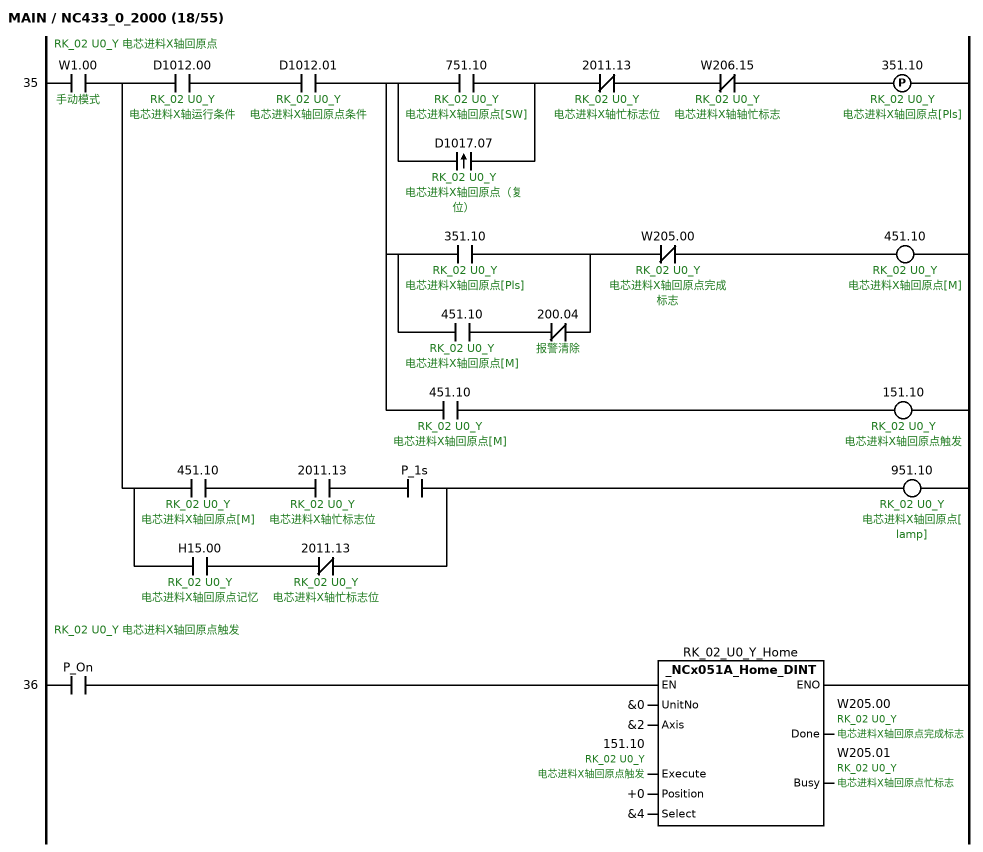
; [picture p72: MAIN / NC433_0_2000, rungs 35-36]
; rung 35: RK_02 U0_Y 电芯进料X轴回原点
LD W1.00  ; 手动模式
OUT TR0
AND D1012.00  ; RK_02 U0_Y 电芯进料X轴运行条件
AND D1012.01  ; RK_02 U0_Y 电芯进料X轴回原点条件
OUT TR1
LD 751.10  ; RK_02 U0_Y 电芯进料X轴回原点[SW]
@OR D1017.07  ; RK_02 U0_Y 电芯进料X轴回原点（复位）
ANDLD
ANDNOT 2011.13  ; RK_02 U0_Y 电芯进料X轴忙标志位
ANDNOT W206.15  ; RK_02 U0_Y 电芯进料X轴轴忙标志
DIFU(013) 351.10  ; RK_02 U0_Y 电芯进料X轴回原点[Pls]
LD TR1
LD 351.10  ; RK_02 U0_Y 电芯进料X轴回原点[Pls]
LD 451.10  ; RK_02 U0_Y 电芯进料X轴回原点[M]
ANDNOT 200.04  ; 报警清除
ORLD
ANDLD
ANDNOT W205.00  ; RK_02 U0_Y 电芯进料X轴回原点完成标志
OUT 451.10  ; RK_02 U0_Y 电芯进料X轴回原点[M]
LD TR1
AND 451.10  ; RK_02 U0_Y 电芯进料X轴回原点[M]
OUT 151.10  ; RK_02 U0_Y 电芯进料X轴回原点触发
LD TR0
LD 451.10  ; RK_02 U0_Y 电芯进料X轴回原点[M]
AND 2011.13  ; RK_02 U0_Y 电芯进料X轴忙标志位
AND P_1s
LD H15.00  ; RK_02 U0_Y 电芯进料X轴回原点记忆
ANDNOT 2011.13  ; RK_02 U0_Y 电芯进料X轴忙标志位
ORLD
ANDLD
OUT 951.10  ; RK_02 U0_Y 电芯进料X轴回原点[lamp]
; rung 36: RK_02 U0_Y 电芯进料X轴回原点触发
LD P_On
CALL RK_02_U0_Y_Home : _NCx051A_Home_DINT (UnitNo := &0, Axis := &2, Execute := 151.10, Position := +0, Select := &4, Done => W205.00, Busy => W205.01)  ; RK_02 U0_Y 电芯进料X轴回原点触发, RK_02 U0_Y 电芯进料X轴回原点完成标志, RK_02 U0_Y 电芯进料X轴回原点忙标志

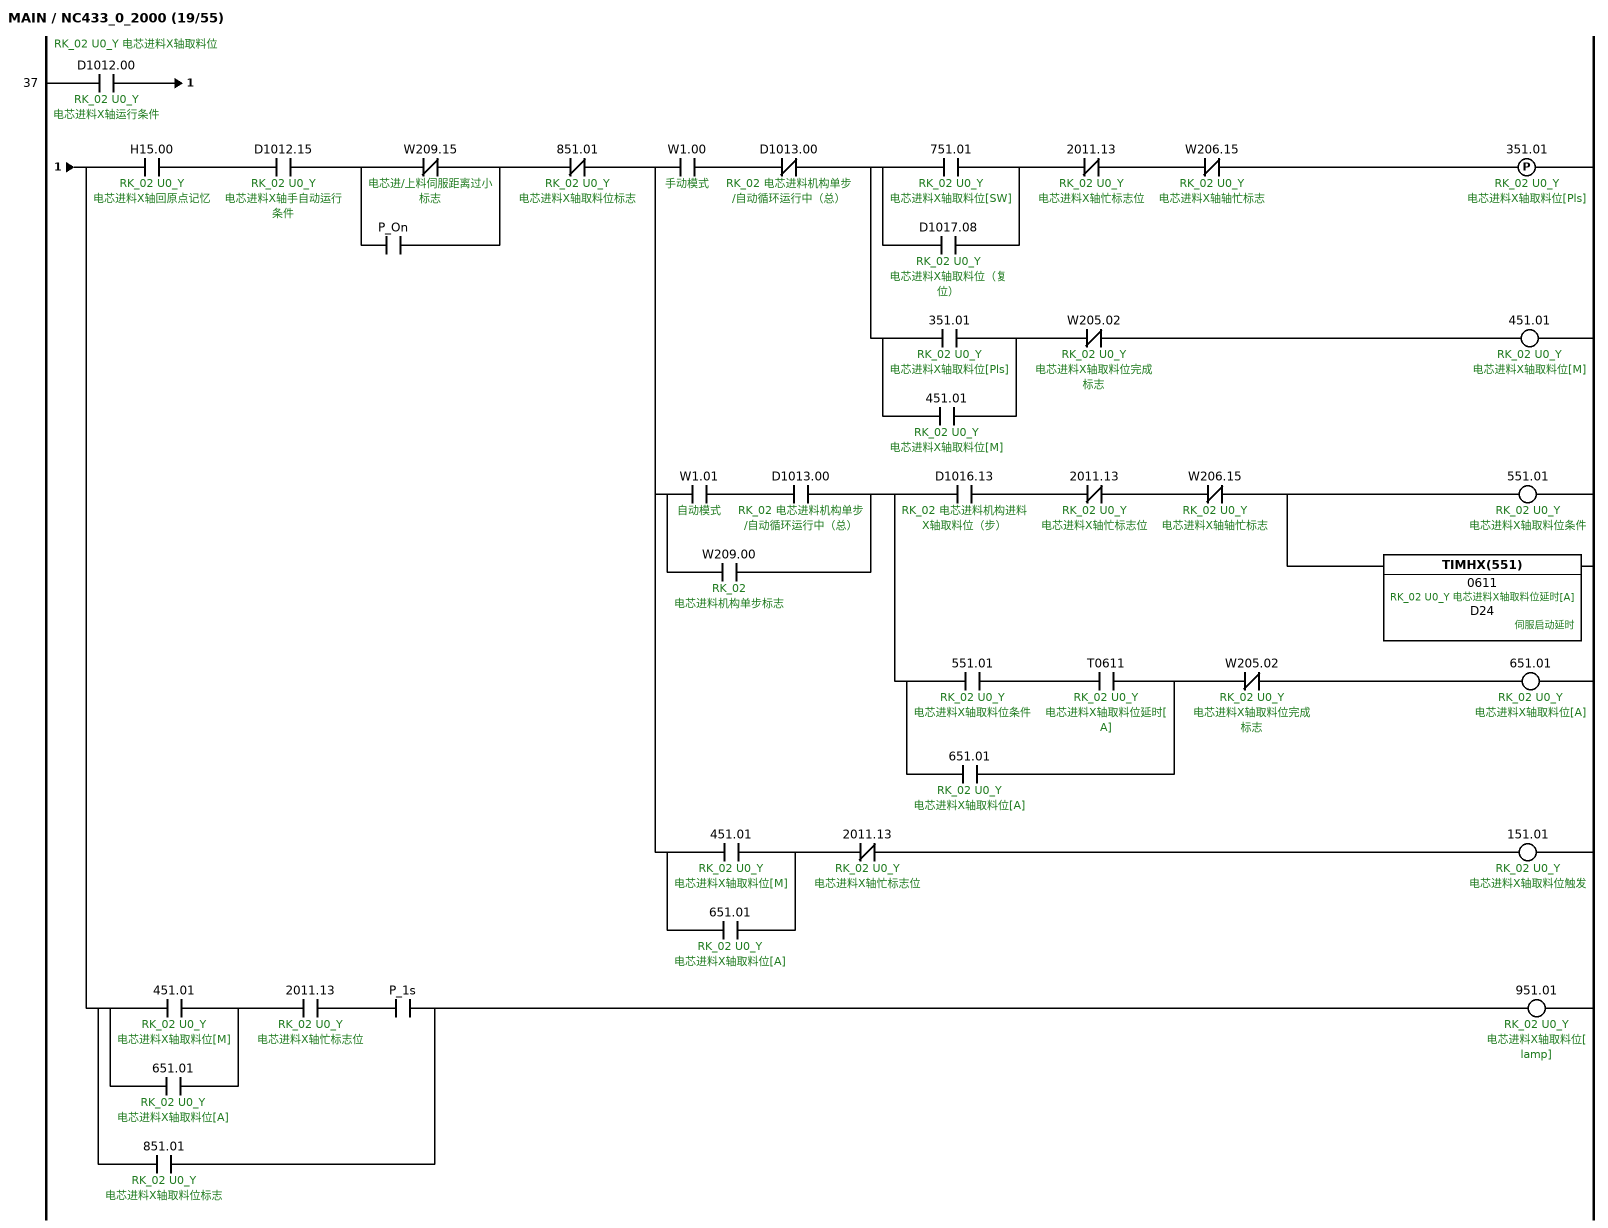
; rung 37: RK_02 U0_Y 电芯进料X轴取料位
LD D1012.00  ; RK_02 U0_Y 电芯进料X轴运行条件
OUT TR0
AND H15.00  ; RK_02 U0_Y 电芯进料X轴回原点记忆
AND D1012.15  ; RK_02 U0_Y 电芯进料X轴手自动运行条件
LDNOT W209.15  ; 电芯进/上料伺服距离过小标志
OR P_On
ANDLD
ANDNOT 851.01  ; RK_02 U0_Y 电芯进料X轴取料位标志
OUT TR1
AND W1.00  ; 手动模式
ANDNOT D1013.00  ; RK_02 电芯进料机构单步/自动循环运行中（总）
OUT TR2
LD 751.01  ; RK_02 U0_Y 电芯进料X轴取料位[SW]
OR D1017.08  ; RK_02 U0_Y 电芯进料X轴取料位（复位）
ANDLD
ANDNOT 2011.13  ; RK_02 U0_Y 电芯进料X轴忙标志位
ANDNOT W206.15  ; RK_02 U0_Y 电芯进料X轴轴忙标志
DIFU(013) 351.01  ; RK_02 U0_Y 电芯进料X轴取料位[Pls]
LD TR2
LD 351.01  ; RK_02 U0_Y 电芯进料X轴取料位[Pls]
OR 451.01  ; RK_02 U0_Y 电芯进料X轴取料位[M]
ANDLD
ANDNOT W205.02  ; RK_02 U0_Y 电芯进料X轴取料位完成标志
OUT 451.01  ; RK_02 U0_Y 电芯进料X轴取料位[M]
LD TR1
LD W1.01  ; 自动模式
AND D1013.00  ; RK_02 电芯进料机构单步/自动循环运行中（总）
OR W209.00  ; RK_02  电芯进料机构单步标志
ANDLD
OUT TR2
AND D1016.13  ; RK_02 电芯进料机构进料X轴取料位（步）
ANDNOT 2011.13  ; RK_02 U0_Y 电芯进料X轴忙标志位
ANDNOT W206.15  ; RK_02 U0_Y 电芯进料X轴轴忙标志
OUT 551.01  ; RK_02 U0_Y 电芯进料X轴取料位条件
TIMHX(551) 0611 D24  ; 伺服启动延时, RK_02 U0_Y 电芯进料X轴取料位延时[A]
LD TR2
LD 551.01  ; RK_02 U0_Y 电芯进料X轴取料位条件
AND T0611  ; RK_02 U0_Y 电芯进料X轴取料位延时[A]
OR 651.01  ; RK_02 U0_Y 电芯进料X轴取料位[A]
ANDLD
ANDNOT W205.02  ; RK_02 U0_Y 电芯进料X轴取料位完成标志
OUT 651.01  ; RK_02 U0_Y 电芯进料X轴取料位[A]
LD TR1
LD 451.01  ; RK_02 U0_Y 电芯进料X轴取料位[M]
OR 651.01  ; RK_02 U0_Y 电芯进料X轴取料位[A]
ANDLD
ANDNOT 2011.13  ; RK_02 U0_Y 电芯进料X轴忙标志位
OUT 151.01  ; RK_02 U0_Y 电芯进料X轴取料位触发
LD TR0
LD 451.01  ; RK_02 U0_Y 电芯进料X轴取料位[M]
OR 651.01  ; RK_02 U0_Y 电芯进料X轴取料位[A]
AND 2011.13  ; RK_02 U0_Y 电芯进料X轴忙标志位
AND P_1s
OR 851.01  ; RK_02 U0_Y 电芯进料X轴取料位标志
ANDLD
OUT 951.01  ; RK_02 U0_Y 电芯进料X轴取料位[lamp]

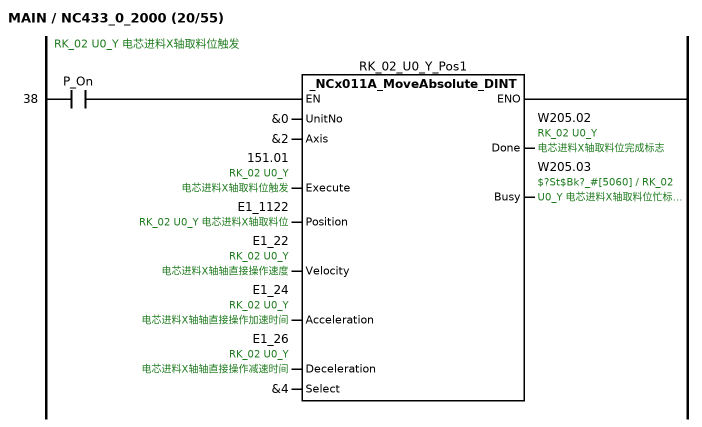
; rung 38: RK_02 U0_Y 电芯进料X轴取料位触发
LD P_On
CALL RK_02_U0_Y_Pos1 : _NCx011A_MoveAbsolute_DINT (UnitNo := &0, Axis := &2, Execute := 151.01, Position := E1_1122, Velocity := E1_22, Acceleration := E1_24, Deceleration := E1_26, Select := &4, Done => W205.02, Busy => W205.03)  ; RK_02 U0_Y 电芯进料X轴取料位触发, RK_02 U0_Y 电芯进料X轴取料位, RK_02 U0_Y 电芯进料X轴轴直接操作速度, RK_02 U0_Y 电芯进料X轴轴直接操作加速时间, RK_02 U0_Y 电芯进料X轴轴直接操作减速时间, RK_02 U0_Y 电芯进料X轴取料位完成标志, $?St$Bk?_#[5060] / RK_02 U0_Y 电芯进料X轴取料位忙标志 / $?St$Bk?_#[5060]

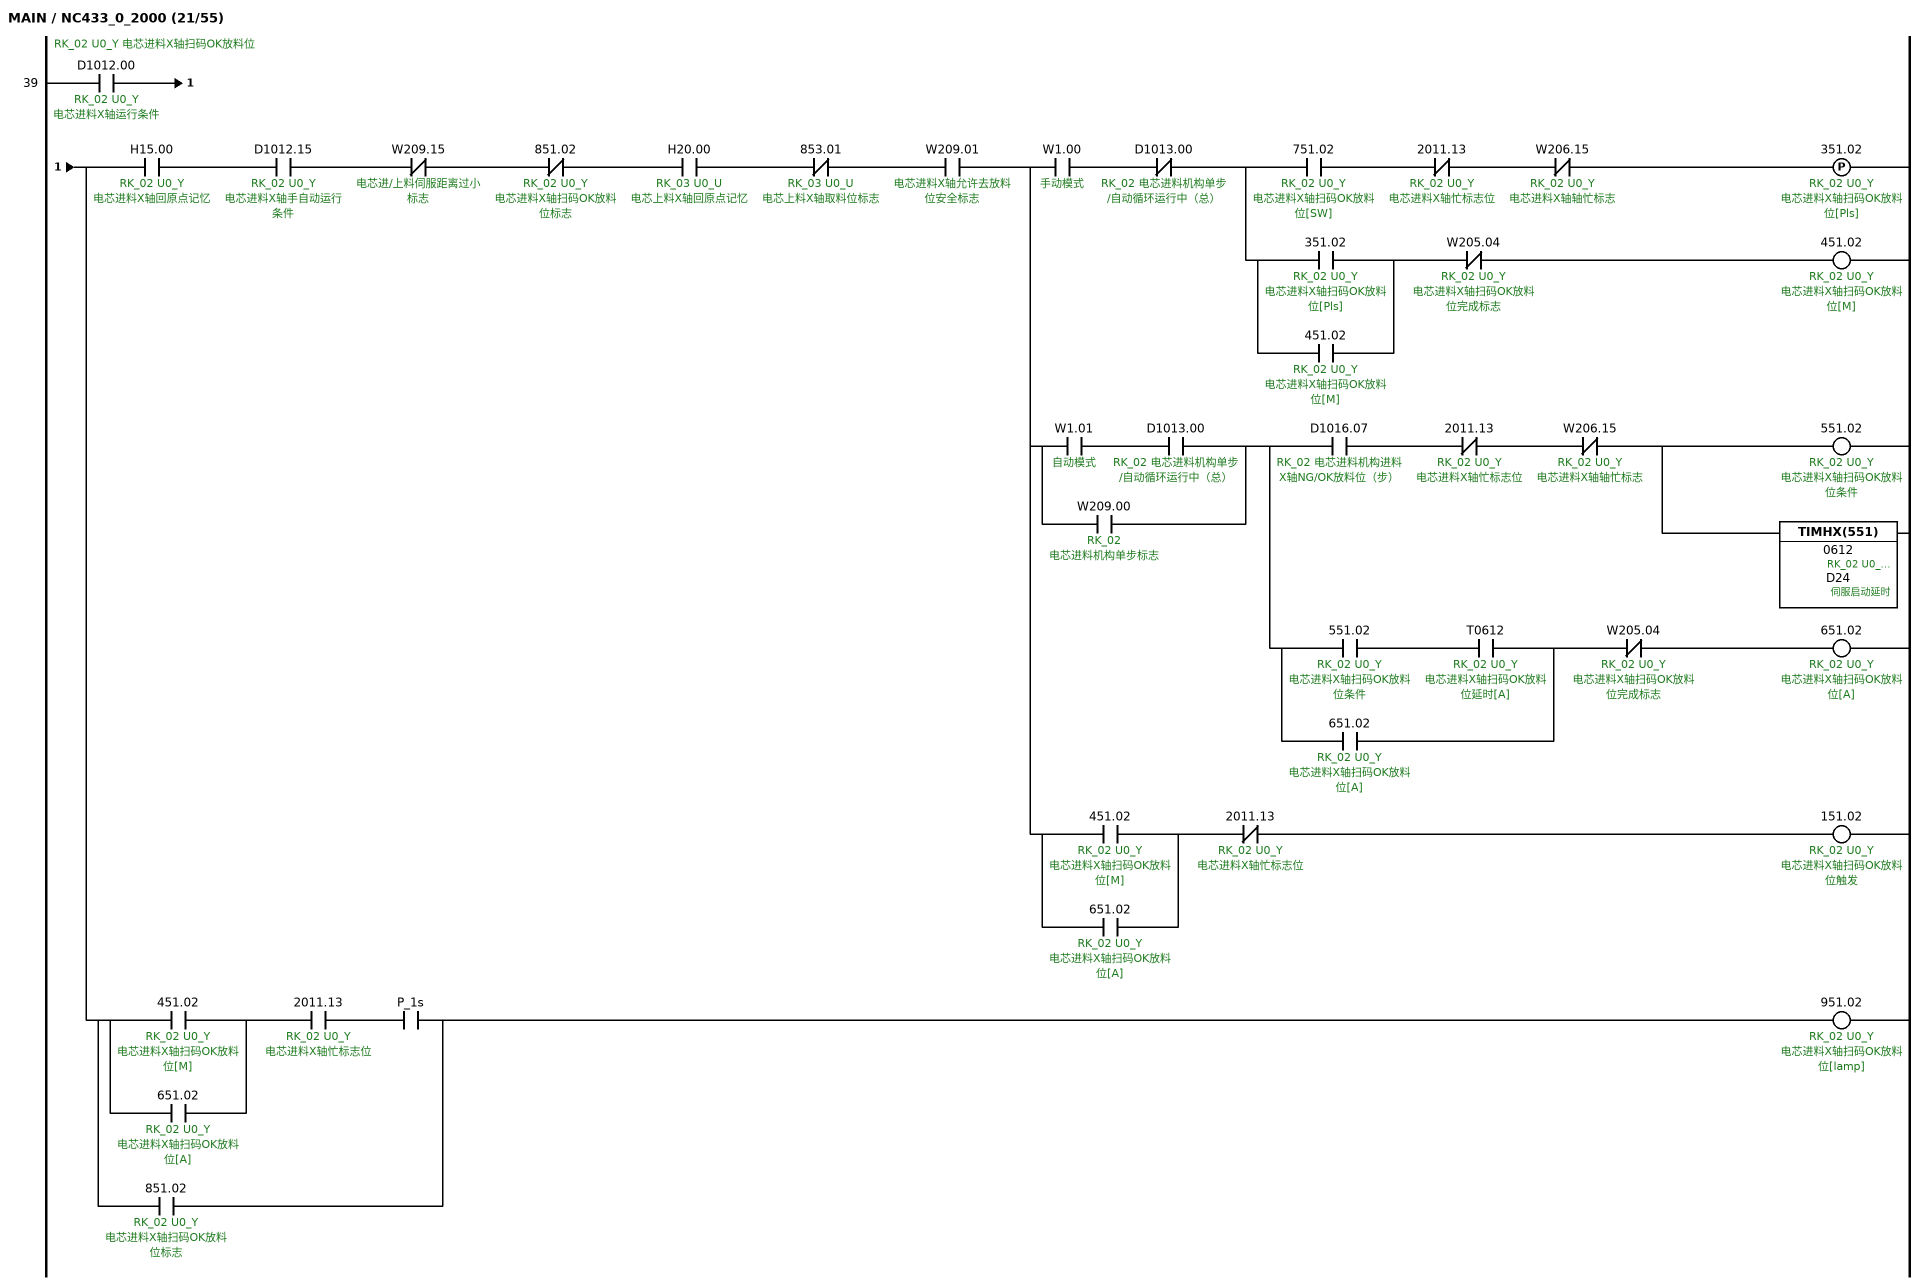
; rung 39: RK_02 U0_Y 电芯进料X轴扫码OK放料位
LD D1012.00  ; RK_02 U0_Y 电芯进料X轴运行条件
OUT TR0
AND H15.00  ; RK_02 U0_Y 电芯进料X轴回原点记忆
AND D1012.15  ; RK_02 U0_Y 电芯进料X轴手自动运行条件
ANDNOT W209.15  ; 电芯进/上料伺服距离过小标志
ANDNOT 851.02  ; RK_02 U0_Y 电芯进料X轴扫码OK放料位标志
AND H20.00  ; RK_03 U0_U 电芯上料X轴回原点记忆
ANDNOT 853.01  ; RK_03 U0_U 电芯上料X轴取料位标志
AND W209.01  ; 电芯进料X轴允许去放料位安全标志
OUT TR1
AND W1.00  ; 手动模式
ANDNOT D1013.00  ; RK_02 电芯进料机构单步/自动循环运行中（总）
OUT TR2
AND 751.02  ; RK_02 U0_Y 电芯进料X轴扫码OK放料位[SW]
ANDNOT 2011.13  ; RK_02 U0_Y 电芯进料X轴忙标志位
ANDNOT W206.15  ; RK_02 U0_Y 电芯进料X轴轴忙标志
DIFU(013) 351.02  ; RK_02 U0_Y 电芯进料X轴扫码OK放料位[Pls]
LD TR2
LD 351.02  ; RK_02 U0_Y 电芯进料X轴扫码OK放料位[Pls]
OR 451.02  ; RK_02 U0_Y 电芯进料X轴扫码OK放料位[M]
ANDLD
ANDNOT W205.04  ; RK_02 U0_Y 电芯进料X轴扫码OK放料位完成标志
OUT 451.02  ; RK_02 U0_Y 电芯进料X轴扫码OK放料位[M]
LD TR1
LD W1.01  ; 自动模式
AND D1013.00  ; RK_02 电芯进料机构单步/自动循环运行中（总）
OR W209.00  ; RK_02  电芯进料机构单步标志
ANDLD
OUT TR2
AND D1016.07  ; RK_02 电芯进料机构进料X轴NG/OK放料位（步）
ANDNOT 2011.13  ; RK_02 U0_Y 电芯进料X轴忙标志位
ANDNOT W206.15  ; RK_02 U0_Y 电芯进料X轴轴忙标志
OUT 551.02  ; RK_02 U0_Y 电芯进料X轴扫码OK放料位条件
TIMHX(551) 0612 D24  ; 伺服启动延时, RK_02 U0_Y 电芯进料X轴扫码OK放料位延时[A]
LD TR2
LD 551.02  ; RK_02 U0_Y 电芯进料X轴扫码OK放料位条件
AND T0612  ; RK_02 U0_Y 电芯进料X轴扫码OK放料位延时[A]
OR 651.02  ; RK_02 U0_Y 电芯进料X轴扫码OK放料位[A]
ANDLD
ANDNOT W205.04  ; RK_02 U0_Y 电芯进料X轴扫码OK放料位完成标志
OUT 651.02  ; RK_02 U0_Y 电芯进料X轴扫码OK放料位[A]
LD TR1
LD 451.02  ; RK_02 U0_Y 电芯进料X轴扫码OK放料位[M]
OR 651.02  ; RK_02 U0_Y 电芯进料X轴扫码OK放料位[A]
ANDLD
ANDNOT 2011.13  ; RK_02 U0_Y 电芯进料X轴忙标志位
OUT 151.02  ; RK_02 U0_Y 电芯进料X轴扫码OK放料位触发
LD TR0
LD 451.02  ; RK_02 U0_Y 电芯进料X轴扫码OK放料位[M]
OR 651.02  ; RK_02 U0_Y 电芯进料X轴扫码OK放料位[A]
AND 2011.13  ; RK_02 U0_Y 电芯进料X轴忙标志位
AND P_1s
OR 851.02  ; RK_02 U0_Y 电芯进料X轴扫码OK放料位标志
ANDLD
OUT 951.02  ; RK_02 U0_Y 电芯进料X轴扫码OK放料位[lamp]

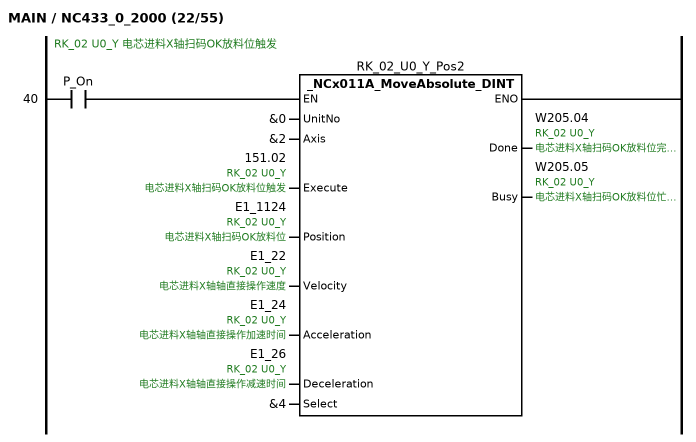
; rung 40: RK_02 U0_Y 电芯进料X轴扫码OK放料位触发
LD P_On
CALL RK_02_U0_Y_Pos2 : _NCx011A_MoveAbsolute_DINT (UnitNo := &0, Axis := &2, Execute := 151.02, Position := E1_1124, Velocity := E1_22, Acceleration := E1_24, Deceleration := E1_26, Select := &4, Done => W205.04, Busy => W205.05)  ; RK_02 U0_Y 电芯进料X轴扫码OK放料位触发, RK_02 U0_Y 电芯进料X轴扫码OK放料位, RK_02 U0_Y 电芯进料X轴轴直接操作速度, RK_02 U0_Y 电芯进料X轴轴直接操作加速时间, RK_02 U0_Y 电芯进料X轴轴直接操作减速时间, RK_02 U0_Y 电芯进料X轴扫码OK放料位完成标志, RK_02 U0_Y 电芯进料X轴扫码OK放料位忙标志

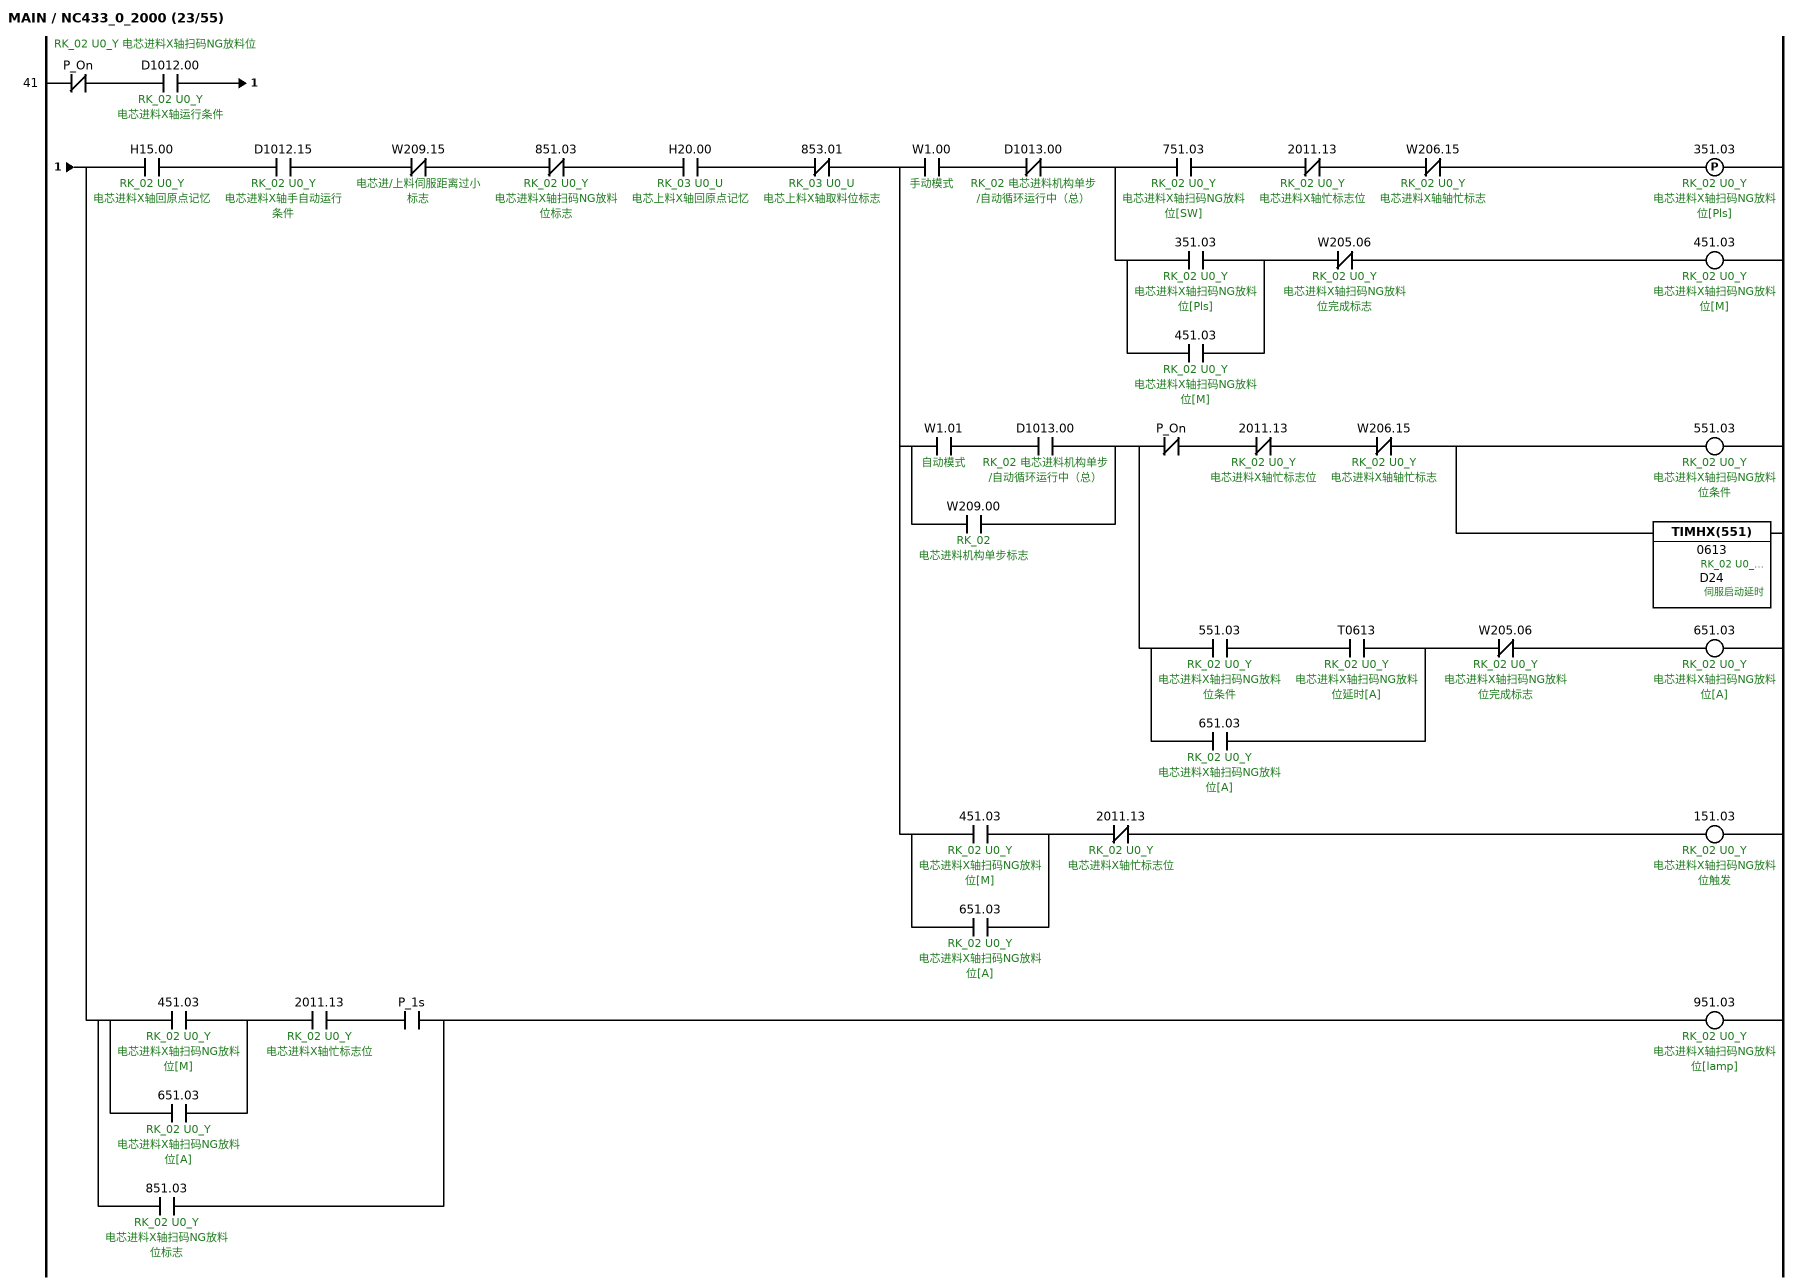
; rung 41: RK_02 U0_Y 电芯进料X轴扫码NG放料位
LDNOT P_On
AND D1012.00  ; RK_02 U0_Y 电芯进料X轴运行条件
OUT TR0
AND H15.00  ; RK_02 U0_Y 电芯进料X轴回原点记忆
AND D1012.15  ; RK_02 U0_Y 电芯进料X轴手自动运行条件
ANDNOT W209.15  ; 电芯进/上料伺服距离过小标志
ANDNOT 851.03  ; RK_02 U0_Y 电芯进料X轴扫码NG放料位标志
AND H20.00  ; RK_03 U0_U 电芯上料X轴回原点记忆
ANDNOT 853.01  ; RK_03 U0_U 电芯上料X轴取料位标志  // 或者改为“RK_03 U0_U 电芯上料X轴当前值”>“最小安全设定值”
OUT TR1
AND W1.00  ; 手动模式
ANDNOT D1013.00  ; RK_02 电芯进料机构单步/自动循环运行中（总）
OUT TR2
AND 751.03  ; RK_02 U0_Y 电芯进料X轴扫码NG放料位[SW]
ANDNOT 2011.13  ; RK_02 U0_Y 电芯进料X轴忙标志位
ANDNOT W206.15  ; RK_02 U0_Y 电芯进料X轴轴忙标志
DIFU(013) 351.03  ; RK_02 U0_Y 电芯进料X轴扫码NG放料位[Pls]
LD TR2
LD 351.03  ; RK_02 U0_Y 电芯进料X轴扫码NG放料位[Pls]
OR 451.03  ; RK_02 U0_Y 电芯进料X轴扫码NG放料位[M]
ANDLD
ANDNOT W205.06  ; RK_02 U0_Y 电芯进料X轴扫码NG放料位完成标志
OUT 451.03  ; RK_02 U0_Y 电芯进料X轴扫码NG放料位[M]
LD TR1
LD W1.01  ; 自动模式
AND D1013.00  ; RK_02 电芯进料机构单步/自动循环运行中（总）
OR W209.00  ; RK_02  电芯进料机构单步标志
ANDLD
OUT TR2
ANDNOT P_On  // RK_02 U0_Y 电芯进料X轴扫码NG放料位（步）
ANDNOT 2011.13  ; RK_02 U0_Y 电芯进料X轴忙标志位
ANDNOT W206.15  ; RK_02 U0_Y 电芯进料X轴轴忙标志
OUT 551.03  ; RK_02 U0_Y 电芯进料X轴扫码NG放料位条件
TIMHX(551) 0613 D24  ; 伺服启动延时, RK_02 U0_Y 电芯进料X轴扫码NG放料位延时[A]
LD TR2
LD 551.03  ; RK_02 U0_Y 电芯进料X轴扫码NG放料位条件
AND T0613  ; RK_02 U0_Y 电芯进料X轴扫码NG放料位延时[A]
OR 651.03  ; RK_02 U0_Y 电芯进料X轴扫码NG放料位[A]
ANDLD
ANDNOT W205.06  ; RK_02 U0_Y 电芯进料X轴扫码NG放料位完成标志
OUT 651.03  ; RK_02 U0_Y 电芯进料X轴扫码NG放料位[A]
LD TR1
LD 451.03  ; RK_02 U0_Y 电芯进料X轴扫码NG放料位[M]
OR 651.03  ; RK_02 U0_Y 电芯进料X轴扫码NG放料位[A]
ANDLD
ANDNOT 2011.13  ; RK_02 U0_Y 电芯进料X轴忙标志位
OUT 151.03  ; RK_02 U0_Y 电芯进料X轴扫码NG放料位触发
LD TR0
LD 451.03  ; RK_02 U0_Y 电芯进料X轴扫码NG放料位[M]
OR 651.03  ; RK_02 U0_Y 电芯进料X轴扫码NG放料位[A]
AND 2011.13  ; RK_02 U0_Y 电芯进料X轴忙标志位
AND P_1s
OR 851.03  ; RK_02 U0_Y 电芯进料X轴扫码NG放料位标志
ANDLD
OUT 951.03  ; RK_02 U0_Y 电芯进料X轴扫码NG放料位[lamp]

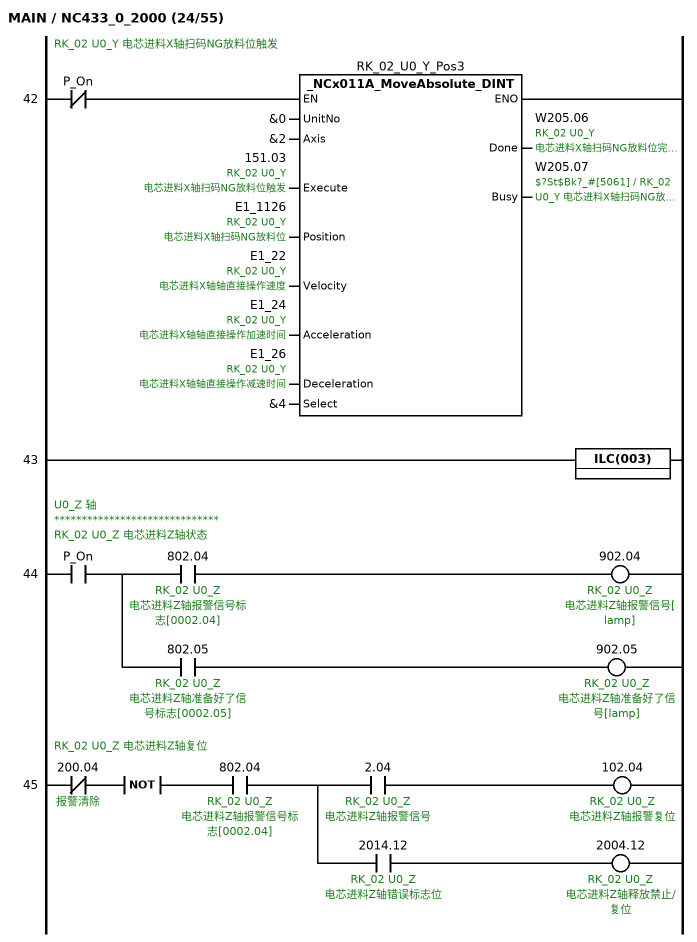
; rung 42: RK_02 U0_Y 电芯进料X轴扫码NG放料位触发
LDNOT P_On
CALL RK_02_U0_Y_Pos3 : _NCx011A_MoveAbsolute_DINT (UnitNo := &0, Axis := &2, Execute := 151.03, Position := E1_1126, Velocity := E1_22, Acceleration := E1_24, Deceleration := E1_26, Select := &4, Done => W205.06, Busy => W205.07)  ; RK_02 U0_Y 电芯进料X轴扫码NG放料位触发, RK_02 U0_Y 电芯进料X轴扫码NG放料位, RK_02 U0_Y 电芯进料X轴轴直接操作速度, RK_02 U0_Y 电芯进料X轴轴直接操作加速时间, RK_02 U0_Y 电芯进料X轴轴直接操作减速时间, RK_02 U0_Y 电芯进料X轴扫码NG放料位完成标志, $?St$Bk?_#[5061] / RK_02 U0_Y 电芯进料X轴扫码NG放料位忙标志 / $?St$Bk?_#[5061]
; rung 43
ILC(003)
; rung 44: U0_Z 轴 / ****************************** / RK_02 U0_Z 电芯进料Z轴状态
LD P_On
OUT TR0
AND 802.04  ; RK_02 U0_Z 电芯进料Z轴报警信号标志[0002.04]
OUT 902.04  ; RK_02 U0_Z 电芯进料Z轴报警信号[lamp]
LD TR0
AND 802.05  ; RK_02 U0_Z 电芯进料Z轴准备好了信号标志[0002.05]
OUT 902.05  ; RK_02 U0_Z 电芯进料Z轴准备好了信号[lamp]
; rung 45: RK_02 U0_Z 电芯进料Z轴复位
LDNOT 200.04  ; 报警清除
NOT(520)
AND 802.04  ; RK_02 U0_Z 电芯进料Z轴报警信号标志[0002.04]
OUT TR0
AND 2.04  ; RK_02 U0_Z 电芯进料Z轴报警信号
OUT 102.04  ; RK_02 U0_Z 电芯进料Z轴报警复位
LD TR0
AND 2014.12  ; RK_02 U0_Z 电芯进料Z轴错误标志位
OUT 2004.12  ; RK_02 U0_Z 电芯进料Z轴释放禁止/复位

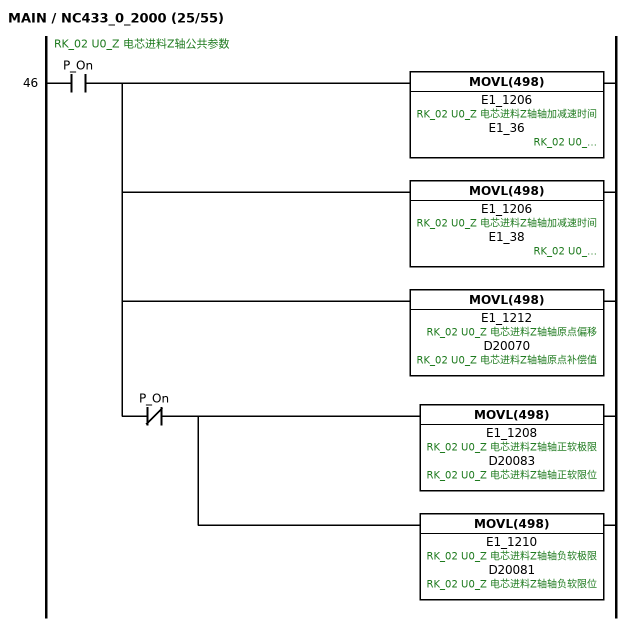
; rung 46: RK_02 U0_Z 电芯进料Z轴公共参数
LD P_On
MOVL(498) E1_1206 E1_36  ; RK_02 U0_Z 电芯进料Z轴轴加减速时间, RK_02 U0_Z 电芯进料Z轴轴直接操作加速时间
MOVL(498) E1_1206 E1_38  ; RK_02 U0_Z 电芯进料Z轴轴加减速时间, RK_02 U0_Z 电芯进料Z轴轴直接操作减速时间
MOVL(498) E1_1212 D20070  ; RK_02 U0_Z 电芯进料Z轴轴原点偏移, RK_02 U0_Z 电芯进料Z轴轴原点补偿值
ANDNOT P_On
MOVL(498) E1_1208 D20083  ; RK_02 U0_Z 电芯进料Z轴轴正软极限, RK_02 U0_Z 电芯进料Z轴轴正软限位
MOVL(498) E1_1210 D20081  ; RK_02 U0_Z 电芯进料Z轴轴负软极限, RK_02 U0_Z 电芯进料Z轴轴负软限位

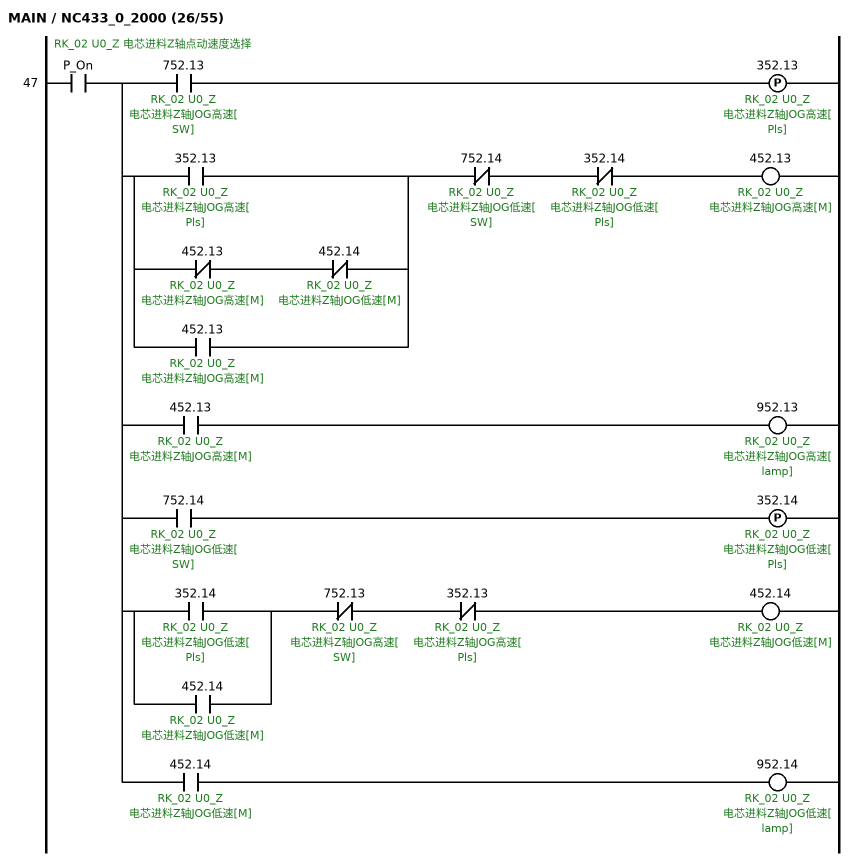
; rung 47: RK_02 U0_Z 电芯进料Z轴点动速度选择
LD P_On
OUT TR0
AND 752.13  ; RK_02 U0_Z 电芯进料Z轴JOG高速[SW]
DIFU(013) 352.13  ; RK_02 U0_Z 电芯进料Z轴JOG高速[Pls]
LD TR0
LD 352.13  ; RK_02 U0_Z 电芯进料Z轴JOG高速[Pls]
LDNOT 452.13  ; RK_02 U0_Z 电芯进料Z轴JOG高速[M]
ANDNOT 452.14  ; RK_02 U0_Z 电芯进料Z轴JOG低速[M]
ORLD
OR 452.13  ; RK_02 U0_Z 电芯进料Z轴JOG高速[M]
ANDLD
ANDNOT 752.14  ; RK_02 U0_Z 电芯进料Z轴JOG低速[SW]
ANDNOT 352.14  ; RK_02 U0_Z 电芯进料Z轴JOG低速[Pls]
OUT 452.13  ; RK_02 U0_Z 电芯进料Z轴JOG高速[M]
LD TR0
AND 452.13  ; RK_02 U0_Z 电芯进料Z轴JOG高速[M]
OUT 952.13  ; RK_02 U0_Z 电芯进料Z轴JOG高速[lamp]
LD TR0
AND 752.14  ; RK_02 U0_Z 电芯进料Z轴JOG低速[SW]
DIFU(013) 352.14  ; RK_02 U0_Z 电芯进料Z轴JOG低速[Pls]
LD TR0
LD 352.14  ; RK_02 U0_Z 电芯进料Z轴JOG低速[Pls]
OR 452.14  ; RK_02 U0_Z 电芯进料Z轴JOG低速[M]
ANDLD
ANDNOT 752.13  ; RK_02 U0_Z 电芯进料Z轴JOG高速[SW]
ANDNOT 352.13  ; RK_02 U0_Z 电芯进料Z轴JOG高速[Pls]
OUT 452.14  ; RK_02 U0_Z 电芯进料Z轴JOG低速[M]
LD TR0
AND 452.14  ; RK_02 U0_Z 电芯进料Z轴JOG低速[M]
OUT 952.14  ; RK_02 U0_Z 电芯进料Z轴JOG低速[lamp]

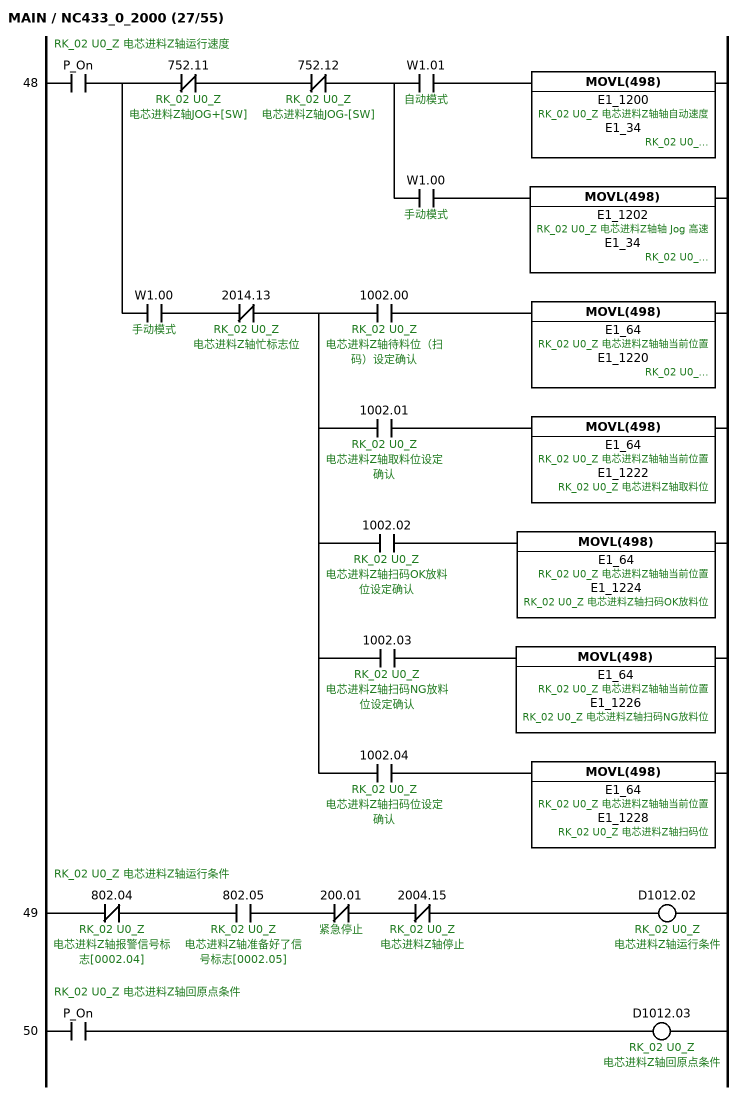
; rung 48: RK_02 U0_Z 电芯进料Z轴运行速度
LD P_On
OUT TR0
ANDNOT 752.11  ; RK_02 U0_Z 电芯进料Z轴JOG+[SW]
ANDNOT 752.12  ; RK_02 U0_Z 电芯进料Z轴JOG-[SW]
OUT TR1
AND W1.01  ; 自动模式
MOVL(498) E1_1200 E1_34  ; RK_02 U0_Z 电芯进料Z轴轴自动速度, RK_02 U0_Z 电芯进料Z轴轴直接操作速度
LD TR1
AND W1.00  ; 手动模式
MOVL(498) E1_1202 E1_34  ; RK_02 U0_Z 电芯进料Z轴轴 Jog 高速, RK_02 U0_Z 电芯进料Z轴轴直接操作速度
LD TR0
AND W1.00  ; 手动模式
ANDNOT 2014.13  ; RK_02 U0_Z 电芯进料Z轴忙标志位
OUT TR0
AND 1002.00  ; RK_02 U0_Z 电芯进料Z轴待料位（扫码）设定确认
MOVL(498) E1_64 E1_1220  ; RK_02 U0_Z 电芯进料Z轴轴当前位置, RK_02 U0_Z 电芯进料Z轴待料位（扫码）
LD TR0
AND 1002.01  ; RK_02 U0_Z 电芯进料Z轴取料位设定确认
MOVL(498) E1_64 E1_1222  ; RK_02 U0_Z 电芯进料Z轴轴当前位置, RK_02 U0_Z 电芯进料Z轴取料位
LD TR0
AND 1002.02  ; RK_02 U0_Z 电芯进料Z轴扫码OK放料位设定确认
MOVL(498) E1_64 E1_1224  ; RK_02 U0_Z 电芯进料Z轴轴当前位置, RK_02 U0_Z 电芯进料Z轴扫码OK放料位
LD TR0
AND 1002.03  ; RK_02 U0_Z 电芯进料Z轴扫码NG放料位设定确认
MOVL(498) E1_64 E1_1226  ; RK_02 U0_Z 电芯进料Z轴轴当前位置, RK_02 U0_Z 电芯进料Z轴扫码NG放料位
LD TR0
AND 1002.04  ; RK_02 U0_Z 电芯进料Z轴扫码位设定确认
MOVL(498) E1_64 E1_1228  ; RK_02 U0_Z 电芯进料Z轴轴当前位置, RK_02 U0_Z 电芯进料Z轴扫码位
; rung 49: RK_02 U0_Z 电芯进料Z轴运行条件
LDNOT 802.04  ; RK_02 U0_Z 电芯进料Z轴报警信号标志[0002.04]
AND 802.05  ; RK_02 U0_Z 电芯进料Z轴准备好了信号标志[0002.05]
ANDNOT 200.01  ; 紧急停止
ANDNOT 2004.15  ; RK_02 U0_Z 电芯进料Z轴停止
OUT D1012.02  ; RK_02 U0_Z 电芯进料Z轴运行条件
; rung 50: RK_02 U0_Z 电芯进料Z轴回原点条件
LD P_On
OUT D1012.03  ; RK_02 U0_Z 电芯进料Z轴回原点条件

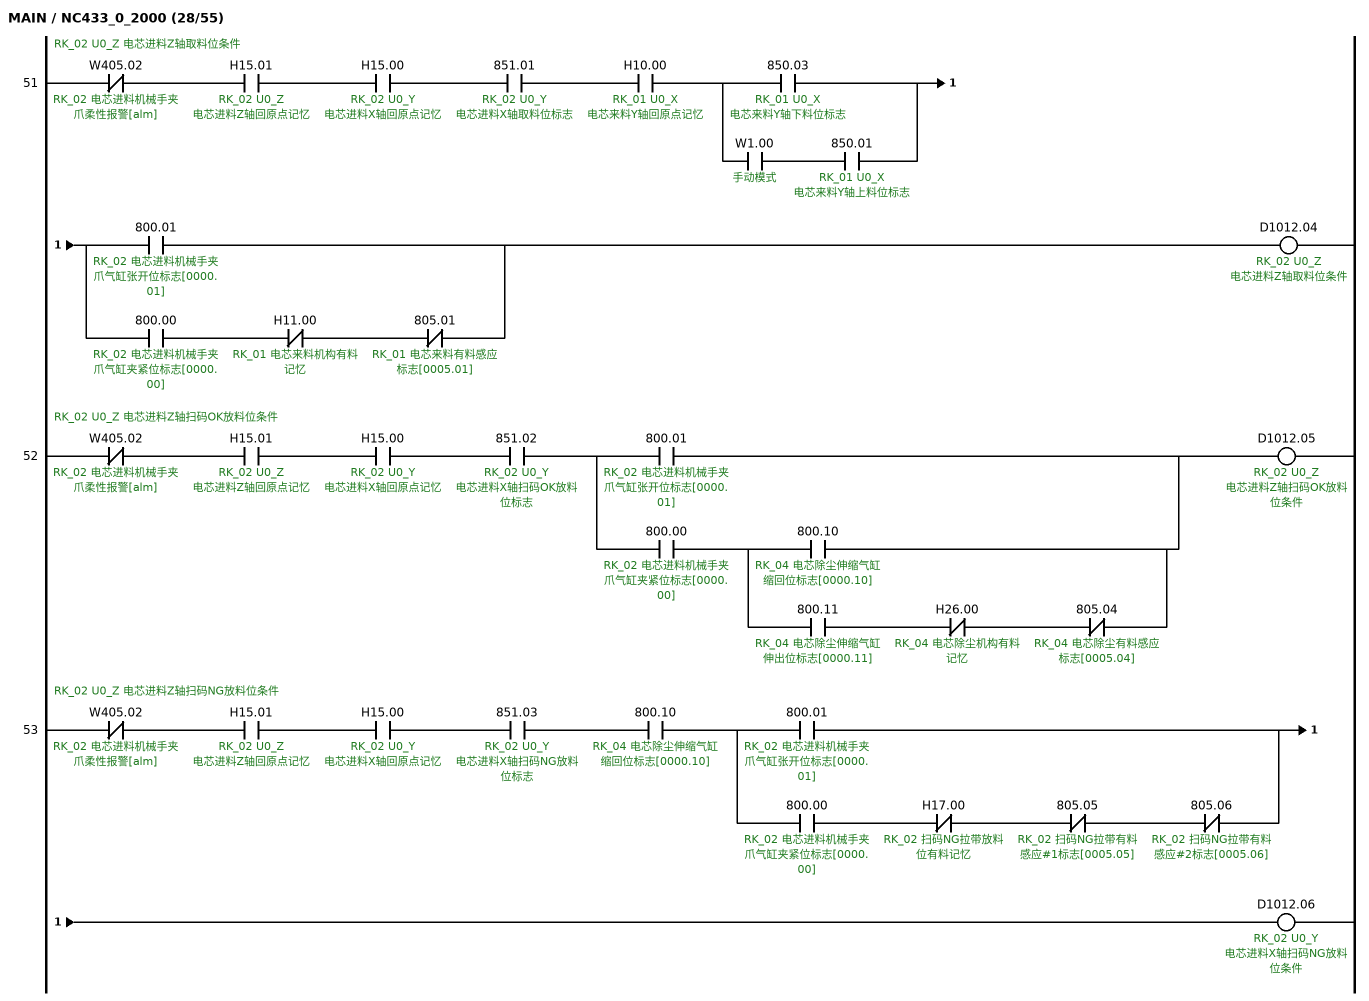
; rung 51: RK_02 U0_Z 电芯进料Z轴取料位条件
LDNOT W405.02  ; RK_02 电芯进料机械手夹爪柔性报警[alm]
AND H15.01  ; RK_02 U0_Z 电芯进料Z轴回原点记忆
AND H15.00  ; RK_02 U0_Y 电芯进料X轴回原点记忆
AND 851.01  ; RK_02 U0_Y 电芯进料X轴取料位标志
AND H10.00  ; RK_01 U0_X 电芯来料Y轴回原点记忆
LD 850.03  ; RK_01 U0_X 电芯来料Y轴下料位标志
LD W1.00  ; 手动模式
AND 850.01  ; RK_01 U0_X 电芯来料Y轴上料位标志
ORLD
ANDLD
LD 800.01  ; RK_02 电芯进料机械手夹爪气缸张开位标志[0000.01]
LD 800.00  ; RK_02 电芯进料机械手夹爪气缸夹紧位标志[0000.00]
ANDNOT H11.00  ; RK_01 电芯来料机构有料记忆
ANDNOT 805.01  ; RK_01 电芯来料有料感应标志[0005.01]
ORLD
ANDLD
OUT D1012.04  ; RK_02 U0_Z 电芯进料Z轴取料位条件
; rung 52: RK_02 U0_Z 电芯进料Z轴扫码OK放料位条件
LDNOT W405.02  ; RK_02 电芯进料机械手夹爪柔性报警[alm]
AND H15.01  ; RK_02 U0_Z 电芯进料Z轴回原点记忆
AND H15.00  ; RK_02 U0_Y 电芯进料X轴回原点记忆
AND 851.02  ; RK_02 U0_Y 电芯进料X轴扫码OK放料位标志
LD 800.01  ; RK_02 电芯进料机械手夹爪气缸张开位标志[0000.01]
LD 800.00  ; RK_02 电芯进料机械手夹爪气缸夹紧位标志[0000.00]
LD 800.10  ; RK_04 电芯除尘伸缩气缸缩回位标志[0000.10]
LD 800.11  ; RK_04 电芯除尘伸缩气缸伸出位标志[0000.11]
ANDNOT H26.00  ; RK_04 电芯除尘机构有料记忆
ANDNOT 805.04  ; RK_04 电芯除尘有料感应标志[0005.04]
ORLD
ANDLD
ORLD
ANDLD
OUT D1012.05  ; RK_02 U0_Z 电芯进料Z轴扫码OK放料位条件
; rung 53: RK_02 U0_Z 电芯进料Z轴扫码NG放料位条件
LDNOT W405.02  ; RK_02 电芯进料机械手夹爪柔性报警[alm]
AND H15.01  ; RK_02 U0_Z 电芯进料Z轴回原点记忆
AND H15.00  ; RK_02 U0_Y 电芯进料X轴回原点记忆
AND 851.03  ; RK_02 U0_Y 电芯进料X轴扫码NG放料位标志
AND 800.10  ; RK_04 电芯除尘伸缩气缸缩回位标志[0000.10]
LD 800.01  ; RK_02 电芯进料机械手夹爪气缸张开位标志[0000.01]
LD 800.00  ; RK_02 电芯进料机械手夹爪气缸夹紧位标志[0000.00]
ANDNOT H17.00  ; RK_02 扫码NG拉带放料位有料记忆
ANDNOT 805.05  ; RK_02 扫码NG拉带有料感应#1标志[0005.05]
ANDNOT 805.06  ; RK_02 扫码NG拉带有料感应#2标志[0005.06]
ORLD
ANDLD
OUT D1012.06  ; RK_02 U0_Y 电芯进料X轴扫码NG放料位条件

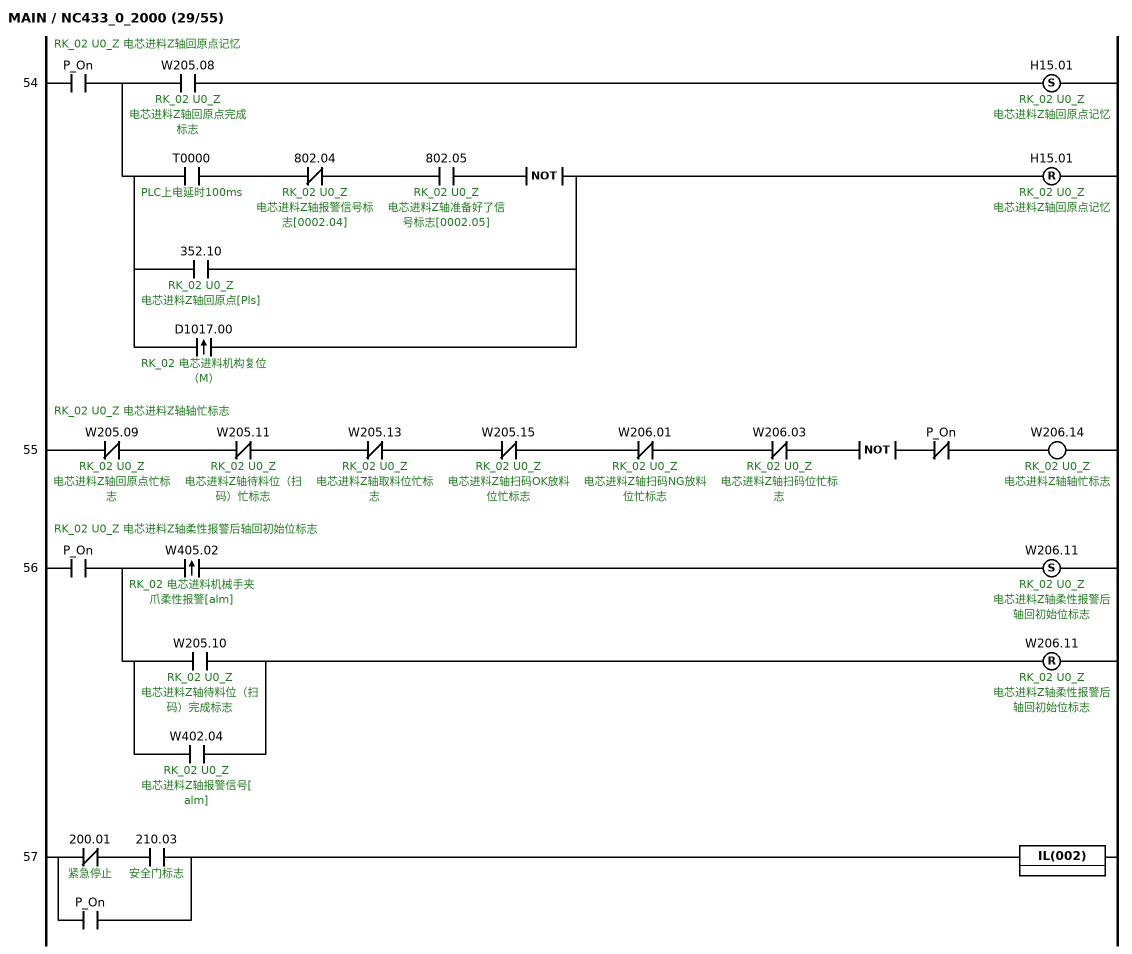
; rung 54: RK_02 U0_Z 电芯进料Z轴回原点记忆
LD P_On
OUT TR0
AND W205.08  ; RK_02 U0_Z 电芯进料Z轴回原点完成标志
SET H15.01  ; RK_02 U0_Z 电芯进料Z轴回原点记忆
LD TR0
LD T0000  ; PLC上电延时100ms
ANDNOT 802.04  ; RK_02 U0_Z 电芯进料Z轴报警信号标志[0002.04]
AND 802.05  ; RK_02 U0_Z 电芯进料Z轴准备好了信号标志[0002.05]
NOT(520)
OR 352.10  ; RK_02 U0_Z 电芯进料Z轴回原点[Pls]
@OR D1017.00  ; RK_02 电芯进料机构复位（M）
ANDLD
RSET H15.01  ; RK_02 U0_Z 电芯进料Z轴回原点记忆
; rung 55: RK_02 U0_Z 电芯进料Z轴轴忙标志
LDNOT W205.09  ; RK_02 U0_Z 电芯进料Z轴回原点忙标志
ANDNOT W205.11  ; RK_02 U0_Z 电芯进料Z轴待料位（扫码）忙标志
ANDNOT W205.13  ; RK_02 U0_Z 电芯进料Z轴取料位忙标志
ANDNOT W205.15  ; RK_02 U0_Z 电芯进料Z轴扫码OK放料位忙标志
ANDNOT W206.01  ; RK_02 U0_Z 电芯进料Z轴扫码NG放料位忙标志
ANDNOT W206.03  ; RK_02 U0_Z 电芯进料Z轴扫码位忙标志
NOT(520)
ANDNOT P_On
OUT W206.14  ; RK_02 U0_Z 电芯进料Z轴轴忙标志
; rung 56: RK_02 U0_Z 电芯进料Z轴柔性报警后轴回初始位标志
LD P_On
OUT TR0
@AND W405.02  ; RK_02 电芯进料机械手夹爪柔性报警[alm]
SET W206.11  ; RK_02 U0_Z 电芯进料Z轴柔性报警后轴回初始位标志
LD TR0
LD W205.10  ; RK_02 U0_Z 电芯进料Z轴待料位（扫码）完成标志
OR W402.04  ; RK_02 U0_Z 电芯进料Z轴报警信号[alm]
ANDLD
RSET W206.11  ; RK_02 U0_Z 电芯进料Z轴柔性报警后轴回初始位标志
; rung 57
LDNOT 200.01  ; 紧急停止
AND 210.03  ; 安全门标志
OR P_On
IL(002)

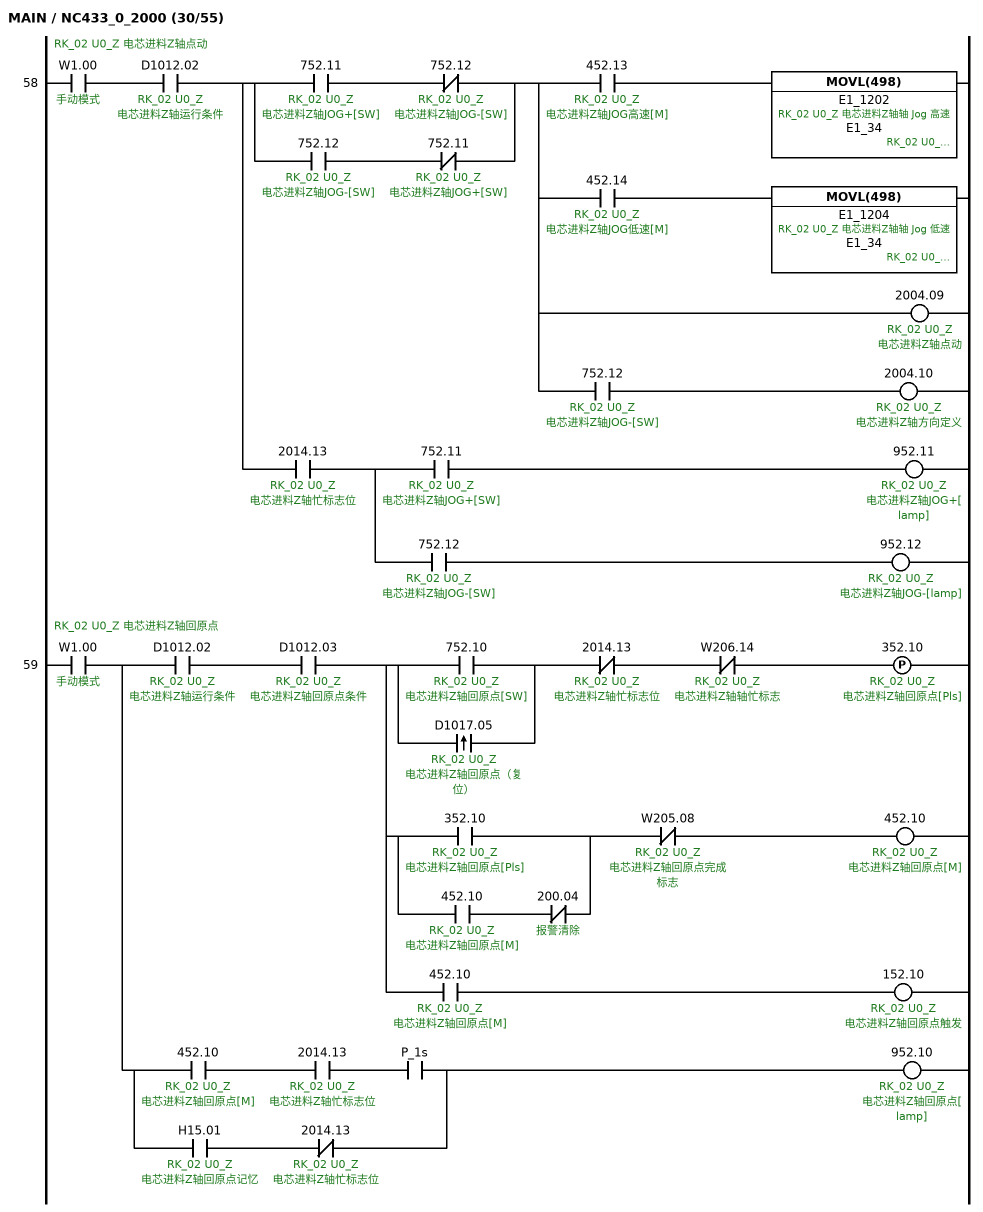
; rung 58: RK_02 U0_Z 电芯进料Z轴点动
LD W1.00  ; 手动模式
AND D1012.02  ; RK_02 U0_Z 电芯进料Z轴运行条件
OUT TR0
LD 752.11  ; RK_02 U0_Z 电芯进料Z轴JOG+[SW]
ANDNOT 752.12  ; RK_02 U0_Z 电芯进料Z轴JOG-[SW]
LD 752.12  ; RK_02 U0_Z 电芯进料Z轴JOG-[SW]
ANDNOT 752.11  ; RK_02 U0_Z 电芯进料Z轴JOG+[SW]
ORLD
ANDLD
OUT TR1
AND 452.13  ; RK_02 U0_Z 电芯进料Z轴JOG高速[M]
MOVL(498) E1_1202 E1_34  ; RK_02 U0_Z 电芯进料Z轴轴 Jog 高速, RK_02 U0_Z 电芯进料Z轴轴直接操作速度
LD TR1
AND 452.14  ; RK_02 U0_Z 电芯进料Z轴JOG低速[M]
MOVL(498) E1_1204 E1_34  ; RK_02 U0_Z 电芯进料Z轴轴 Jog 低速, RK_02 U0_Z 电芯进料Z轴轴直接操作速度
LD TR1
OUT 2004.09  ; RK_02 U0_Z 电芯进料Z轴点动
AND 752.12  ; RK_02 U0_Z 电芯进料Z轴JOG-[SW]
OUT 2004.10  ; RK_02 U0_Z 电芯进料Z轴方向定义
LD TR0
AND 2014.13  ; RK_02 U0_Z 电芯进料Z轴忙标志位
OUT TR0
AND 752.11  ; RK_02 U0_Z 电芯进料Z轴JOG+[SW]
OUT 952.11  ; RK_02 U0_Z 电芯进料Z轴JOG+[lamp]
LD TR0
AND 752.12  ; RK_02 U0_Z 电芯进料Z轴JOG-[SW]
OUT 952.12  ; RK_02 U0_Z 电芯进料Z轴JOG-[lamp]
; rung 59: RK_02 U0_Z 电芯进料Z轴回原点
LD W1.00  ; 手动模式
OUT TR0
AND D1012.02  ; RK_02 U0_Z 电芯进料Z轴运行条件
AND D1012.03  ; RK_02 U0_Z 电芯进料Z轴回原点条件
OUT TR1
LD 752.10  ; RK_02 U0_Z 电芯进料Z轴回原点[SW]
@OR D1017.05  ; RK_02 U0_Z 电芯进料Z轴回原点（复位）
ANDLD
ANDNOT 2014.13  ; RK_02 U0_Z 电芯进料Z轴忙标志位
ANDNOT W206.14  ; RK_02 U0_Z 电芯进料Z轴轴忙标志
DIFU(013) 352.10  ; RK_02 U0_Z 电芯进料Z轴回原点[Pls]
LD TR1
LD 352.10  ; RK_02 U0_Z 电芯进料Z轴回原点[Pls]
LD 452.10  ; RK_02 U0_Z 电芯进料Z轴回原点[M]
ANDNOT 200.04  ; 报警清除
ORLD
ANDLD
ANDNOT W205.08  ; RK_02 U0_Z 电芯进料Z轴回原点完成标志
OUT 452.10  ; RK_02 U0_Z 电芯进料Z轴回原点[M]
LD TR1
AND 452.10  ; RK_02 U0_Z 电芯进料Z轴回原点[M]
OUT 152.10  ; RK_02 U0_Z 电芯进料Z轴回原点触发
LD TR0
LD 452.10  ; RK_02 U0_Z 电芯进料Z轴回原点[M]
AND 2014.13  ; RK_02 U0_Z 电芯进料Z轴忙标志位
AND P_1s
LD H15.01  ; RK_02 U0_Z 电芯进料Z轴回原点记忆
ANDNOT 2014.13  ; RK_02 U0_Z 电芯进料Z轴忙标志位
ORLD
ANDLD
OUT 952.10  ; RK_02 U0_Z 电芯进料Z轴回原点[lamp]

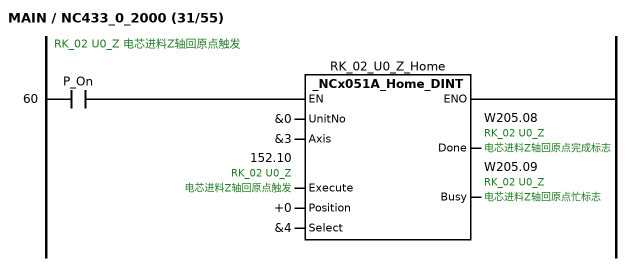
; rung 60: RK_02 U0_Z 电芯进料Z轴回原点触发
LD P_On
CALL RK_02_U0_Z_Home : _NCx051A_Home_DINT (UnitNo := &0, Axis := &3, Execute := 152.10, Position := +0, Select := &4, Done => W205.08, Busy => W205.09)  ; RK_02 U0_Z 电芯进料Z轴回原点触发, RK_02 U0_Z 电芯进料Z轴回原点完成标志, RK_02 U0_Z 电芯进料Z轴回原点忙标志

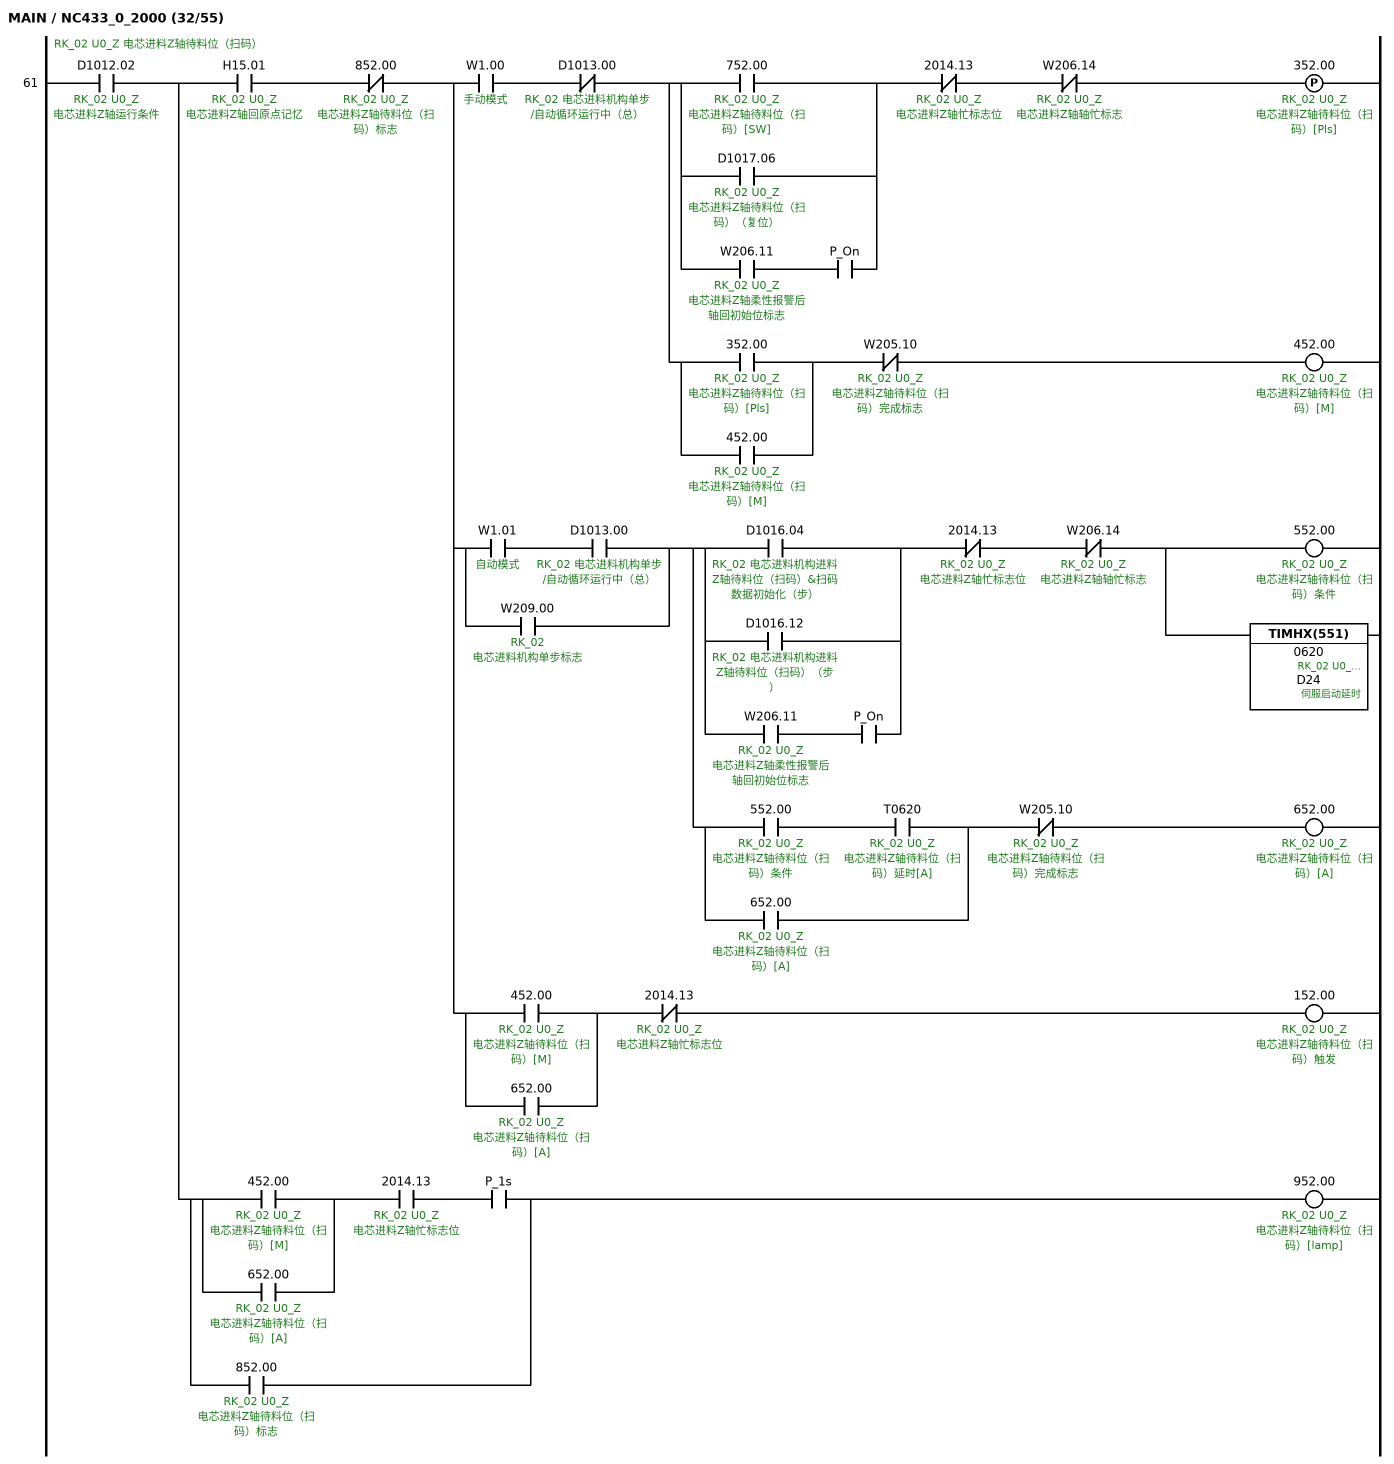
; rung 61: RK_02 U0_Z 电芯进料Z轴待料位（扫码）
LD D1012.02  ; RK_02 U0_Z 电芯进料Z轴运行条件
OUT TR0
AND H15.01  ; RK_02 U0_Z 电芯进料Z轴回原点记忆
ANDNOT 852.00  ; RK_02 U0_Z 电芯进料Z轴待料位（扫码）标志
OUT TR1
AND W1.00  ; 手动模式
ANDNOT D1013.00  ; RK_02 电芯进料机构单步/自动循环运行中（总）
OUT TR2
LD 752.00  ; RK_02 U0_Z 电芯进料Z轴待料位（扫码）[SW]
OR D1017.06  ; RK_02 U0_Z 电芯进料Z轴待料位（扫码）（复位）
LD W206.11  ; RK_02 U0_Z 电芯进料Z轴柔性报警后轴回初始位标志
AND P_On
ORLD
ANDLD
ANDNOT 2014.13  ; RK_02 U0_Z 电芯进料Z轴忙标志位
ANDNOT W206.14  ; RK_02 U0_Z 电芯进料Z轴轴忙标志
DIFU(013) 352.00  ; RK_02 U0_Z 电芯进料Z轴待料位（扫码）[Pls]
LD TR2
LD 352.00  ; RK_02 U0_Z 电芯进料Z轴待料位（扫码）[Pls]
OR 452.00  ; RK_02 U0_Z 电芯进料Z轴待料位（扫码）[M]
ANDLD
ANDNOT W205.10  ; RK_02 U0_Z 电芯进料Z轴待料位（扫码）完成标志
OUT 452.00  ; RK_02 U0_Z 电芯进料Z轴待料位（扫码）[M]
LD TR1
LD W1.01  ; 自动模式
AND D1013.00  ; RK_02 电芯进料机构单步/自动循环运行中（总）
OR W209.00  ; RK_02  电芯进料机构单步标志
ANDLD
OUT TR2
LD D1016.04  ; RK_02 电芯进料机构进料Z轴待料位（扫码）&扫码数据初始化（步）
OR D1016.12  ; RK_02 电芯进料机构进料Z轴待料位（扫码）（步）
LD W206.11  ; RK_02 U0_Z 电芯进料Z轴柔性报警后轴回初始位标志
AND P_On
ORLD
ANDLD
ANDNOT 2014.13  ; RK_02 U0_Z 电芯进料Z轴忙标志位
ANDNOT W206.14  ; RK_02 U0_Z 电芯进料Z轴轴忙标志
OUT 552.00  ; RK_02 U0_Z 电芯进料Z轴待料位（扫码）条件
TIMHX(551) 0620 D24  ; 伺服启动延时, RK_02 U0_Z 电芯进料Z轴待料位（扫码）延时[A]
LD TR2
LD 552.00  ; RK_02 U0_Z 电芯进料Z轴待料位（扫码）条件
AND T0620  ; RK_02 U0_Z 电芯进料Z轴待料位（扫码）延时[A]
OR 652.00  ; RK_02 U0_Z 电芯进料Z轴待料位（扫码）[A]
ANDLD
ANDNOT W205.10  ; RK_02 U0_Z 电芯进料Z轴待料位（扫码）完成标志
OUT 652.00  ; RK_02 U0_Z 电芯进料Z轴待料位（扫码）[A]
LD TR1
LD 452.00  ; RK_02 U0_Z 电芯进料Z轴待料位（扫码）[M]
OR 652.00  ; RK_02 U0_Z 电芯进料Z轴待料位（扫码）[A]
ANDLD
ANDNOT 2014.13  ; RK_02 U0_Z 电芯进料Z轴忙标志位
OUT 152.00  ; RK_02 U0_Z 电芯进料Z轴待料位（扫码）触发
LD TR0
LD 452.00  ; RK_02 U0_Z 电芯进料Z轴待料位（扫码）[M]
OR 652.00  ; RK_02 U0_Z 电芯进料Z轴待料位（扫码）[A]
AND 2014.13  ; RK_02 U0_Z 电芯进料Z轴忙标志位
AND P_1s
OR 852.00  ; RK_02 U0_Z 电芯进料Z轴待料位（扫码）标志
ANDLD
OUT 952.00  ; RK_02 U0_Z 电芯进料Z轴待料位（扫码）[lamp]

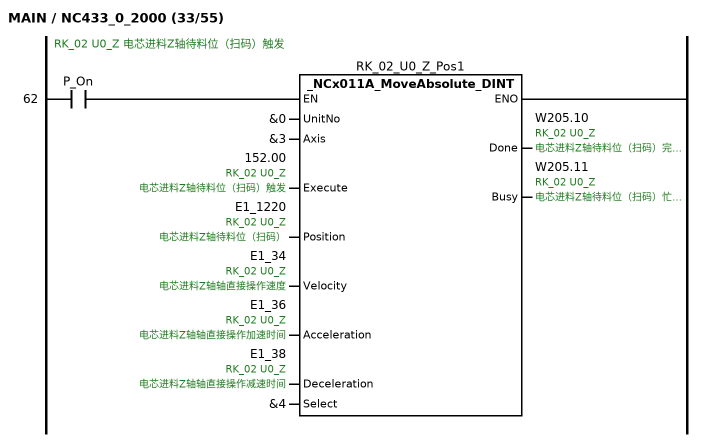
; rung 62: RK_02 U0_Z 电芯进料Z轴待料位（扫码）触发
LD P_On
CALL RK_02_U0_Z_Pos1 : _NCx011A_MoveAbsolute_DINT (UnitNo := &0, Axis := &3, Execute := 152.00, Position := E1_1220, Velocity := E1_34, Acceleration := E1_36, Deceleration := E1_38, Select := &4, Done => W205.10, Busy => W205.11)  ; RK_02 U0_Z 电芯进料Z轴待料位（扫码）触发, RK_02 U0_Z 电芯进料Z轴待料位（扫码）, RK_02 U0_Z 电芯进料Z轴轴直接操作速度, RK_02 U0_Z 电芯进料Z轴轴直接操作加速时间, RK_02 U0_Z 电芯进料Z轴轴直接操作减速时间, RK_02 U0_Z 电芯进料Z轴待料位（扫码）完成标志, RK_02 U0_Z 电芯进料Z轴待料位（扫码）忙标志

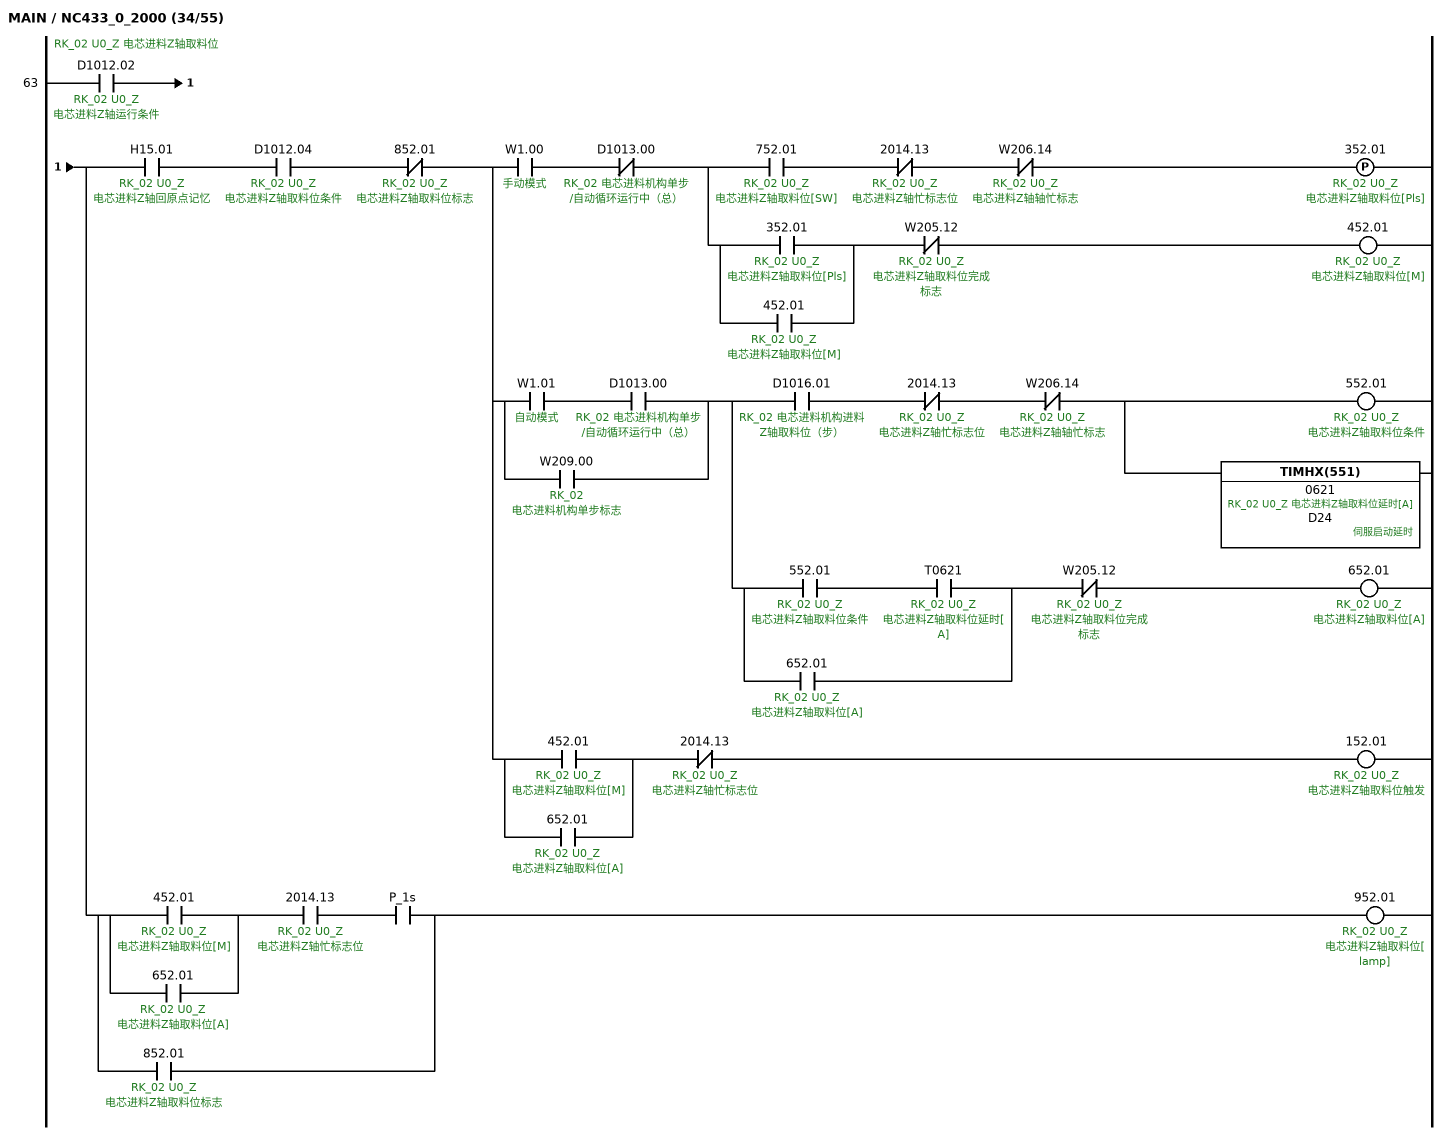
; rung 63: RK_02 U0_Z 电芯进料Z轴取料位
LD D1012.02  ; RK_02 U0_Z 电芯进料Z轴运行条件
OUT TR0
AND H15.01  ; RK_02 U0_Z 电芯进料Z轴回原点记忆
AND D1012.04  ; RK_02 U0_Z 电芯进料Z轴取料位条件
ANDNOT 852.01  ; RK_02 U0_Z 电芯进料Z轴取料位标志
OUT TR1
AND W1.00  ; 手动模式
ANDNOT D1013.00  ; RK_02 电芯进料机构单步/自动循环运行中（总）
OUT TR2
AND 752.01  ; RK_02 U0_Z 电芯进料Z轴取料位[SW]
ANDNOT 2014.13  ; RK_02 U0_Z 电芯进料Z轴忙标志位
ANDNOT W206.14  ; RK_02 U0_Z 电芯进料Z轴轴忙标志
DIFU(013) 352.01  ; RK_02 U0_Z 电芯进料Z轴取料位[Pls]
LD TR2
LD 352.01  ; RK_02 U0_Z 电芯进料Z轴取料位[Pls]
OR 452.01  ; RK_02 U0_Z 电芯进料Z轴取料位[M]
ANDLD
ANDNOT W205.12  ; RK_02 U0_Z 电芯进料Z轴取料位完成标志
OUT 452.01  ; RK_02 U0_Z 电芯进料Z轴取料位[M]
LD TR1
LD W1.01  ; 自动模式
AND D1013.00  ; RK_02 电芯进料机构单步/自动循环运行中（总）
OR W209.00  ; RK_02  电芯进料机构单步标志
ANDLD
OUT TR2
AND D1016.01  ; RK_02 电芯进料机构进料Z轴取料位（步）
ANDNOT 2014.13  ; RK_02 U0_Z 电芯进料Z轴忙标志位
ANDNOT W206.14  ; RK_02 U0_Z 电芯进料Z轴轴忙标志
OUT 552.01  ; RK_02 U0_Z 电芯进料Z轴取料位条件
TIMHX(551) 0621 D24  ; 伺服启动延时, RK_02 U0_Z 电芯进料Z轴取料位延时[A]
LD TR2
LD 552.01  ; RK_02 U0_Z 电芯进料Z轴取料位条件
AND T0621  ; RK_02 U0_Z 电芯进料Z轴取料位延时[A]
OR 652.01  ; RK_02 U0_Z 电芯进料Z轴取料位[A]
ANDLD
ANDNOT W205.12  ; RK_02 U0_Z 电芯进料Z轴取料位完成标志
OUT 652.01  ; RK_02 U0_Z 电芯进料Z轴取料位[A]
LD TR1
LD 452.01  ; RK_02 U0_Z 电芯进料Z轴取料位[M]
OR 652.01  ; RK_02 U0_Z 电芯进料Z轴取料位[A]
ANDLD
ANDNOT 2014.13  ; RK_02 U0_Z 电芯进料Z轴忙标志位
OUT 152.01  ; RK_02 U0_Z 电芯进料Z轴取料位触发
LD TR0
LD 452.01  ; RK_02 U0_Z 电芯进料Z轴取料位[M]
OR 652.01  ; RK_02 U0_Z 电芯进料Z轴取料位[A]
AND 2014.13  ; RK_02 U0_Z 电芯进料Z轴忙标志位
AND P_1s
OR 852.01  ; RK_02 U0_Z 电芯进料Z轴取料位标志
ANDLD
OUT 952.01  ; RK_02 U0_Z 电芯进料Z轴取料位[lamp]

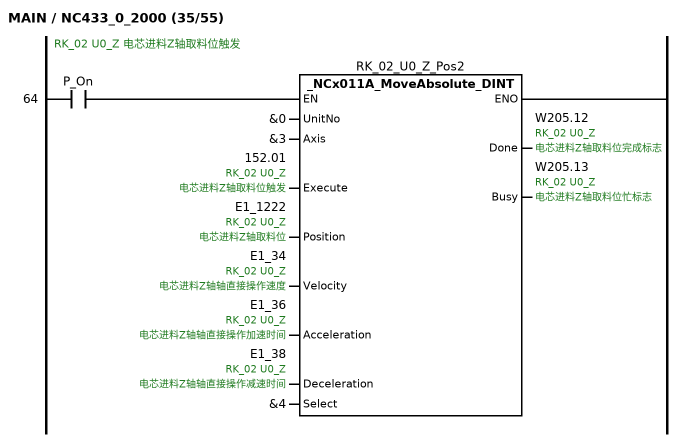
; rung 64: RK_02 U0_Z 电芯进料Z轴取料位触发
LD P_On
CALL RK_02_U0_Z_Pos2 : _NCx011A_MoveAbsolute_DINT (UnitNo := &0, Axis := &3, Execute := 152.01, Position := E1_1222, Velocity := E1_34, Acceleration := E1_36, Deceleration := E1_38, Select := &4, Done => W205.12, Busy => W205.13)  ; RK_02 U0_Z 电芯进料Z轴取料位触发, RK_02 U0_Z 电芯进料Z轴取料位, RK_02 U0_Z 电芯进料Z轴轴直接操作速度, RK_02 U0_Z 电芯进料Z轴轴直接操作加速时间, RK_02 U0_Z 电芯进料Z轴轴直接操作减速时间, RK_02 U0_Z 电芯进料Z轴取料位完成标志, RK_02 U0_Z 电芯进料Z轴取料位忙标志

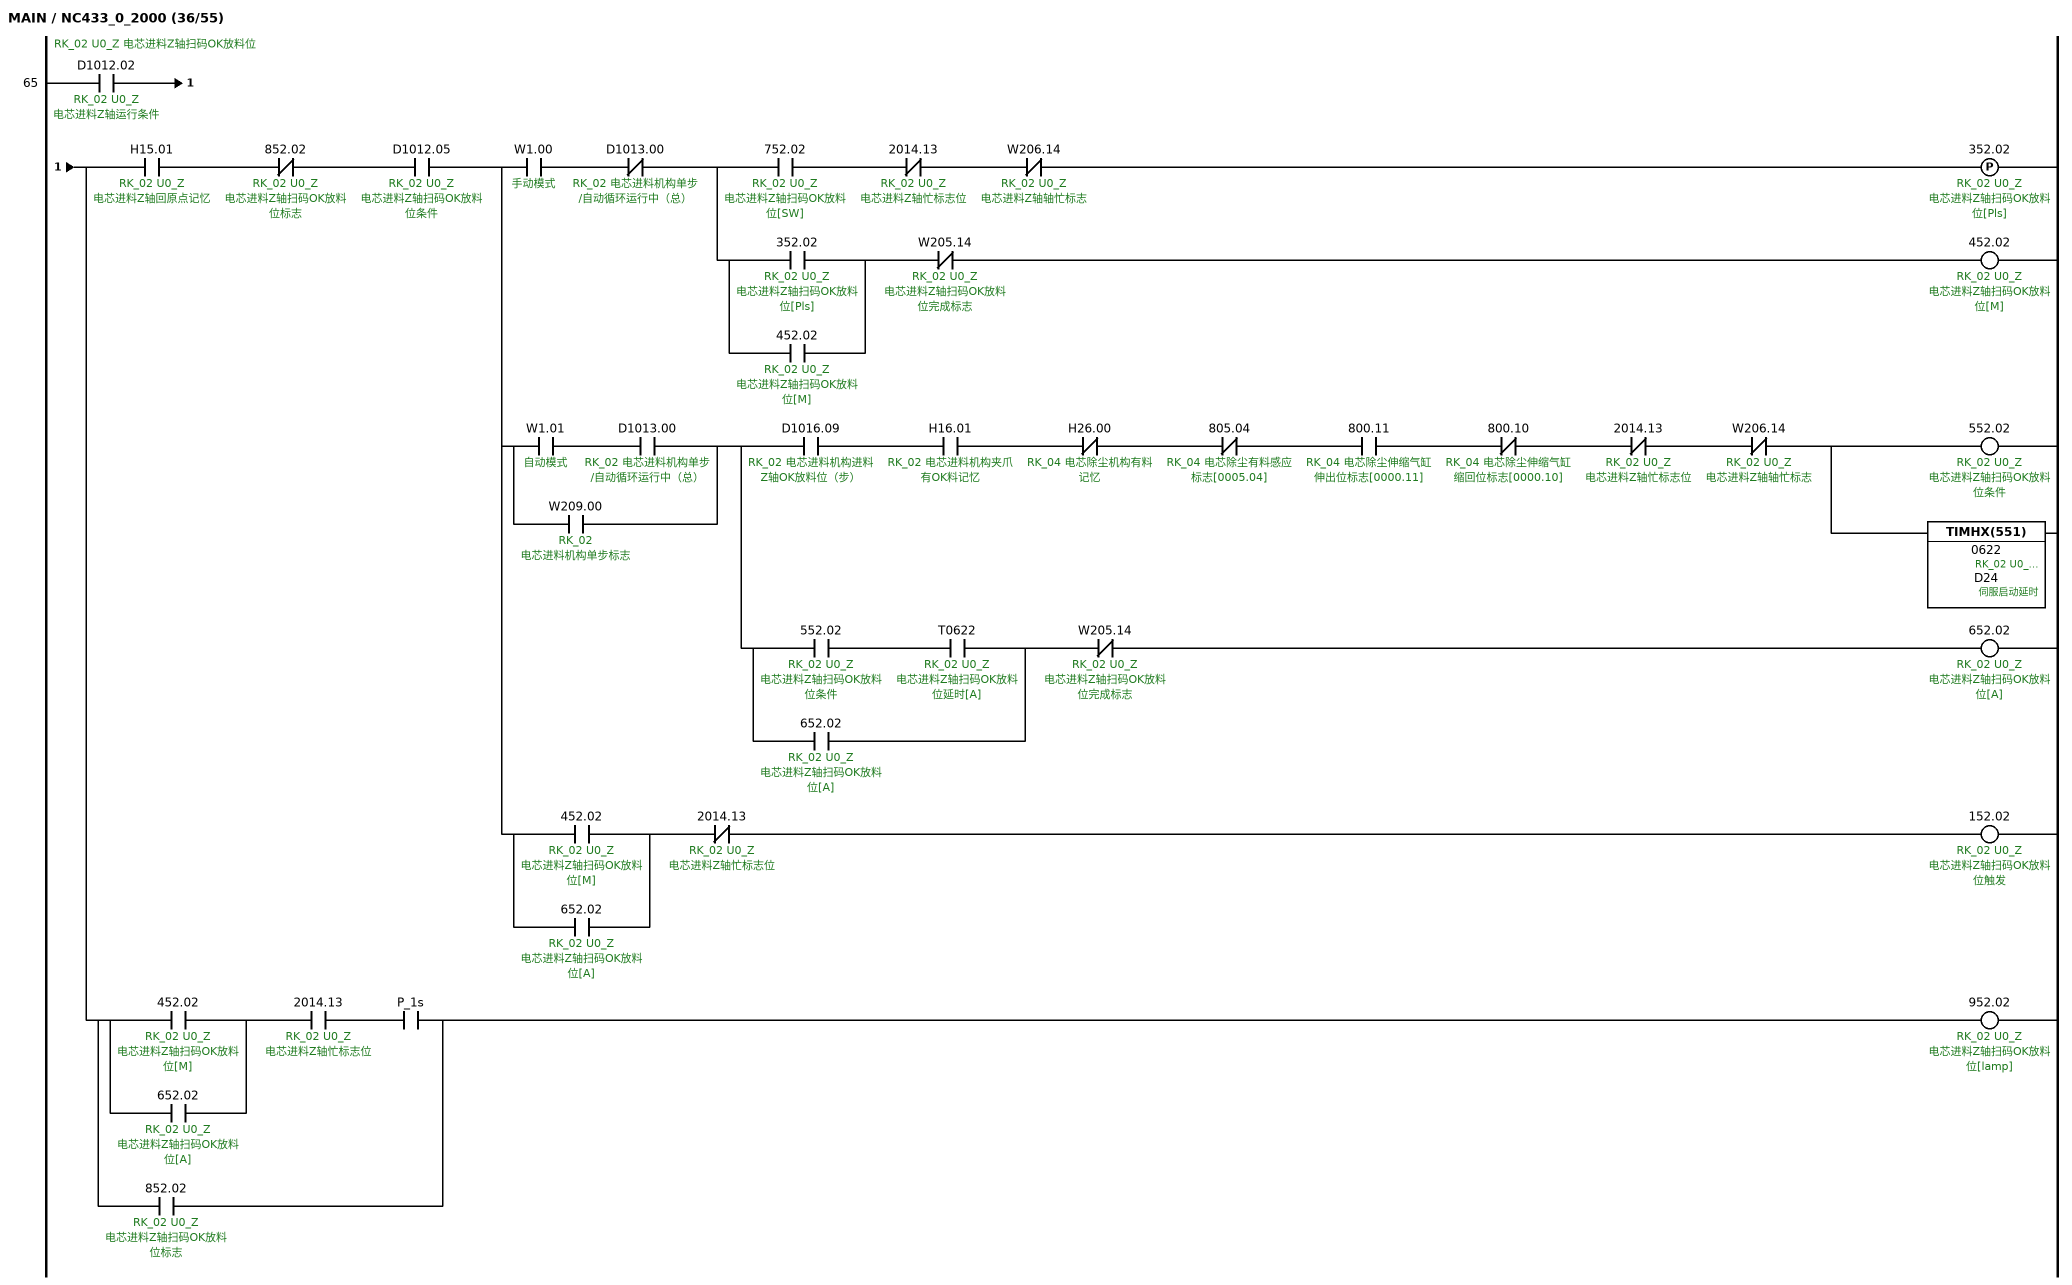
; rung 65: RK_02 U0_Z 电芯进料Z轴扫码OK放料位
LD D1012.02  ; RK_02 U0_Z 电芯进料Z轴运行条件
OUT TR0
AND H15.01  ; RK_02 U0_Z 电芯进料Z轴回原点记忆
ANDNOT 852.02  ; RK_02 U0_Z 电芯进料Z轴扫码OK放料位标志
AND D1012.05  ; RK_02 U0_Z 电芯进料Z轴扫码OK放料位条件
OUT TR1
AND W1.00  ; 手动模式
ANDNOT D1013.00  ; RK_02 电芯进料机构单步/自动循环运行中（总）
OUT TR2
AND 752.02  ; RK_02 U0_Z 电芯进料Z轴扫码OK放料位[SW]
ANDNOT 2014.13  ; RK_02 U0_Z 电芯进料Z轴忙标志位
ANDNOT W206.14  ; RK_02 U0_Z 电芯进料Z轴轴忙标志
DIFU(013) 352.02  ; RK_02 U0_Z 电芯进料Z轴扫码OK放料位[Pls]
LD TR2
LD 352.02  ; RK_02 U0_Z 电芯进料Z轴扫码OK放料位[Pls]
OR 452.02  ; RK_02 U0_Z 电芯进料Z轴扫码OK放料位[M]
ANDLD
ANDNOT W205.14  ; RK_02 U0_Z 电芯进料Z轴扫码OK放料位完成标志
OUT 452.02  ; RK_02 U0_Z 电芯进料Z轴扫码OK放料位[M]
LD TR1
LD W1.01  ; 自动模式
AND D1013.00  ; RK_02 电芯进料机构单步/自动循环运行中（总）
OR W209.00  ; RK_02  电芯进料机构单步标志
ANDLD
OUT TR2
AND D1016.09  ; RK_02 电芯进料机构进料Z轴OK放料位（步）
AND H16.01  ; RK_02 电芯进料机构夹爪有OK料记忆
ANDNOT H26.00  ; RK_04 电芯除尘机构有料记忆
ANDNOT 805.04  ; RK_04 电芯除尘有料感应标志[0005.04]
AND 800.11  ; RK_04 电芯除尘伸缩气缸伸出位标志[0000.11]
ANDNOT 800.10  ; RK_04 电芯除尘伸缩气缸缩回位标志[0000.10]
ANDNOT 2014.13  ; RK_02 U0_Z 电芯进料Z轴忙标志位
ANDNOT W206.14  ; RK_02 U0_Z 电芯进料Z轴轴忙标志
OUT 552.02  ; RK_02 U0_Z 电芯进料Z轴扫码OK放料位条件
TIMHX(551) 0622 D24  ; 伺服启动延时, RK_02 U0_Z 电芯进料Z轴扫码OK放料位延时[A]
LD TR2
LD 552.02  ; RK_02 U0_Z 电芯进料Z轴扫码OK放料位条件
AND T0622  ; RK_02 U0_Z 电芯进料Z轴扫码OK放料位延时[A]
OR 652.02  ; RK_02 U0_Z 电芯进料Z轴扫码OK放料位[A]
ANDLD
ANDNOT W205.14  ; RK_02 U0_Z 电芯进料Z轴扫码OK放料位完成标志
OUT 652.02  ; RK_02 U0_Z 电芯进料Z轴扫码OK放料位[A]
LD TR1
LD 452.02  ; RK_02 U0_Z 电芯进料Z轴扫码OK放料位[M]
OR 652.02  ; RK_02 U0_Z 电芯进料Z轴扫码OK放料位[A]
ANDLD
ANDNOT 2014.13  ; RK_02 U0_Z 电芯进料Z轴忙标志位
OUT 152.02  ; RK_02 U0_Z 电芯进料Z轴扫码OK放料位触发
LD TR0
LD 452.02  ; RK_02 U0_Z 电芯进料Z轴扫码OK放料位[M]
OR 652.02  ; RK_02 U0_Z 电芯进料Z轴扫码OK放料位[A]
AND 2014.13  ; RK_02 U0_Z 电芯进料Z轴忙标志位
AND P_1s
OR 852.02  ; RK_02 U0_Z 电芯进料Z轴扫码OK放料位标志
ANDLD
OUT 952.02  ; RK_02 U0_Z 电芯进料Z轴扫码OK放料位[lamp]

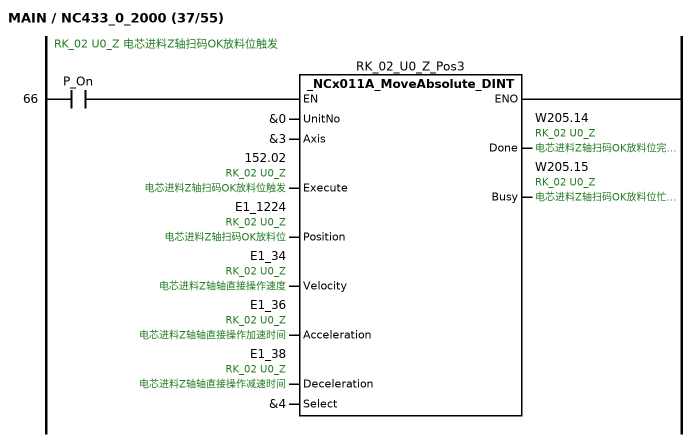
; rung 66: RK_02 U0_Z 电芯进料Z轴扫码OK放料位触发
LD P_On
CALL RK_02_U0_Z_Pos3 : _NCx011A_MoveAbsolute_DINT (UnitNo := &0, Axis := &3, Execute := 152.02, Position := E1_1224, Velocity := E1_34, Acceleration := E1_36, Deceleration := E1_38, Select := &4, Done => W205.14, Busy => W205.15)  ; RK_02 U0_Z 电芯进料Z轴扫码OK放料位触发, RK_02 U0_Z 电芯进料Z轴扫码OK放料位, RK_02 U0_Z 电芯进料Z轴轴直接操作速度, RK_02 U0_Z 电芯进料Z轴轴直接操作加速时间, RK_02 U0_Z 电芯进料Z轴轴直接操作减速时间, RK_02 U0_Z 电芯进料Z轴扫码OK放料位完成标志, RK_02 U0_Z 电芯进料Z轴扫码OK放料位忙标志

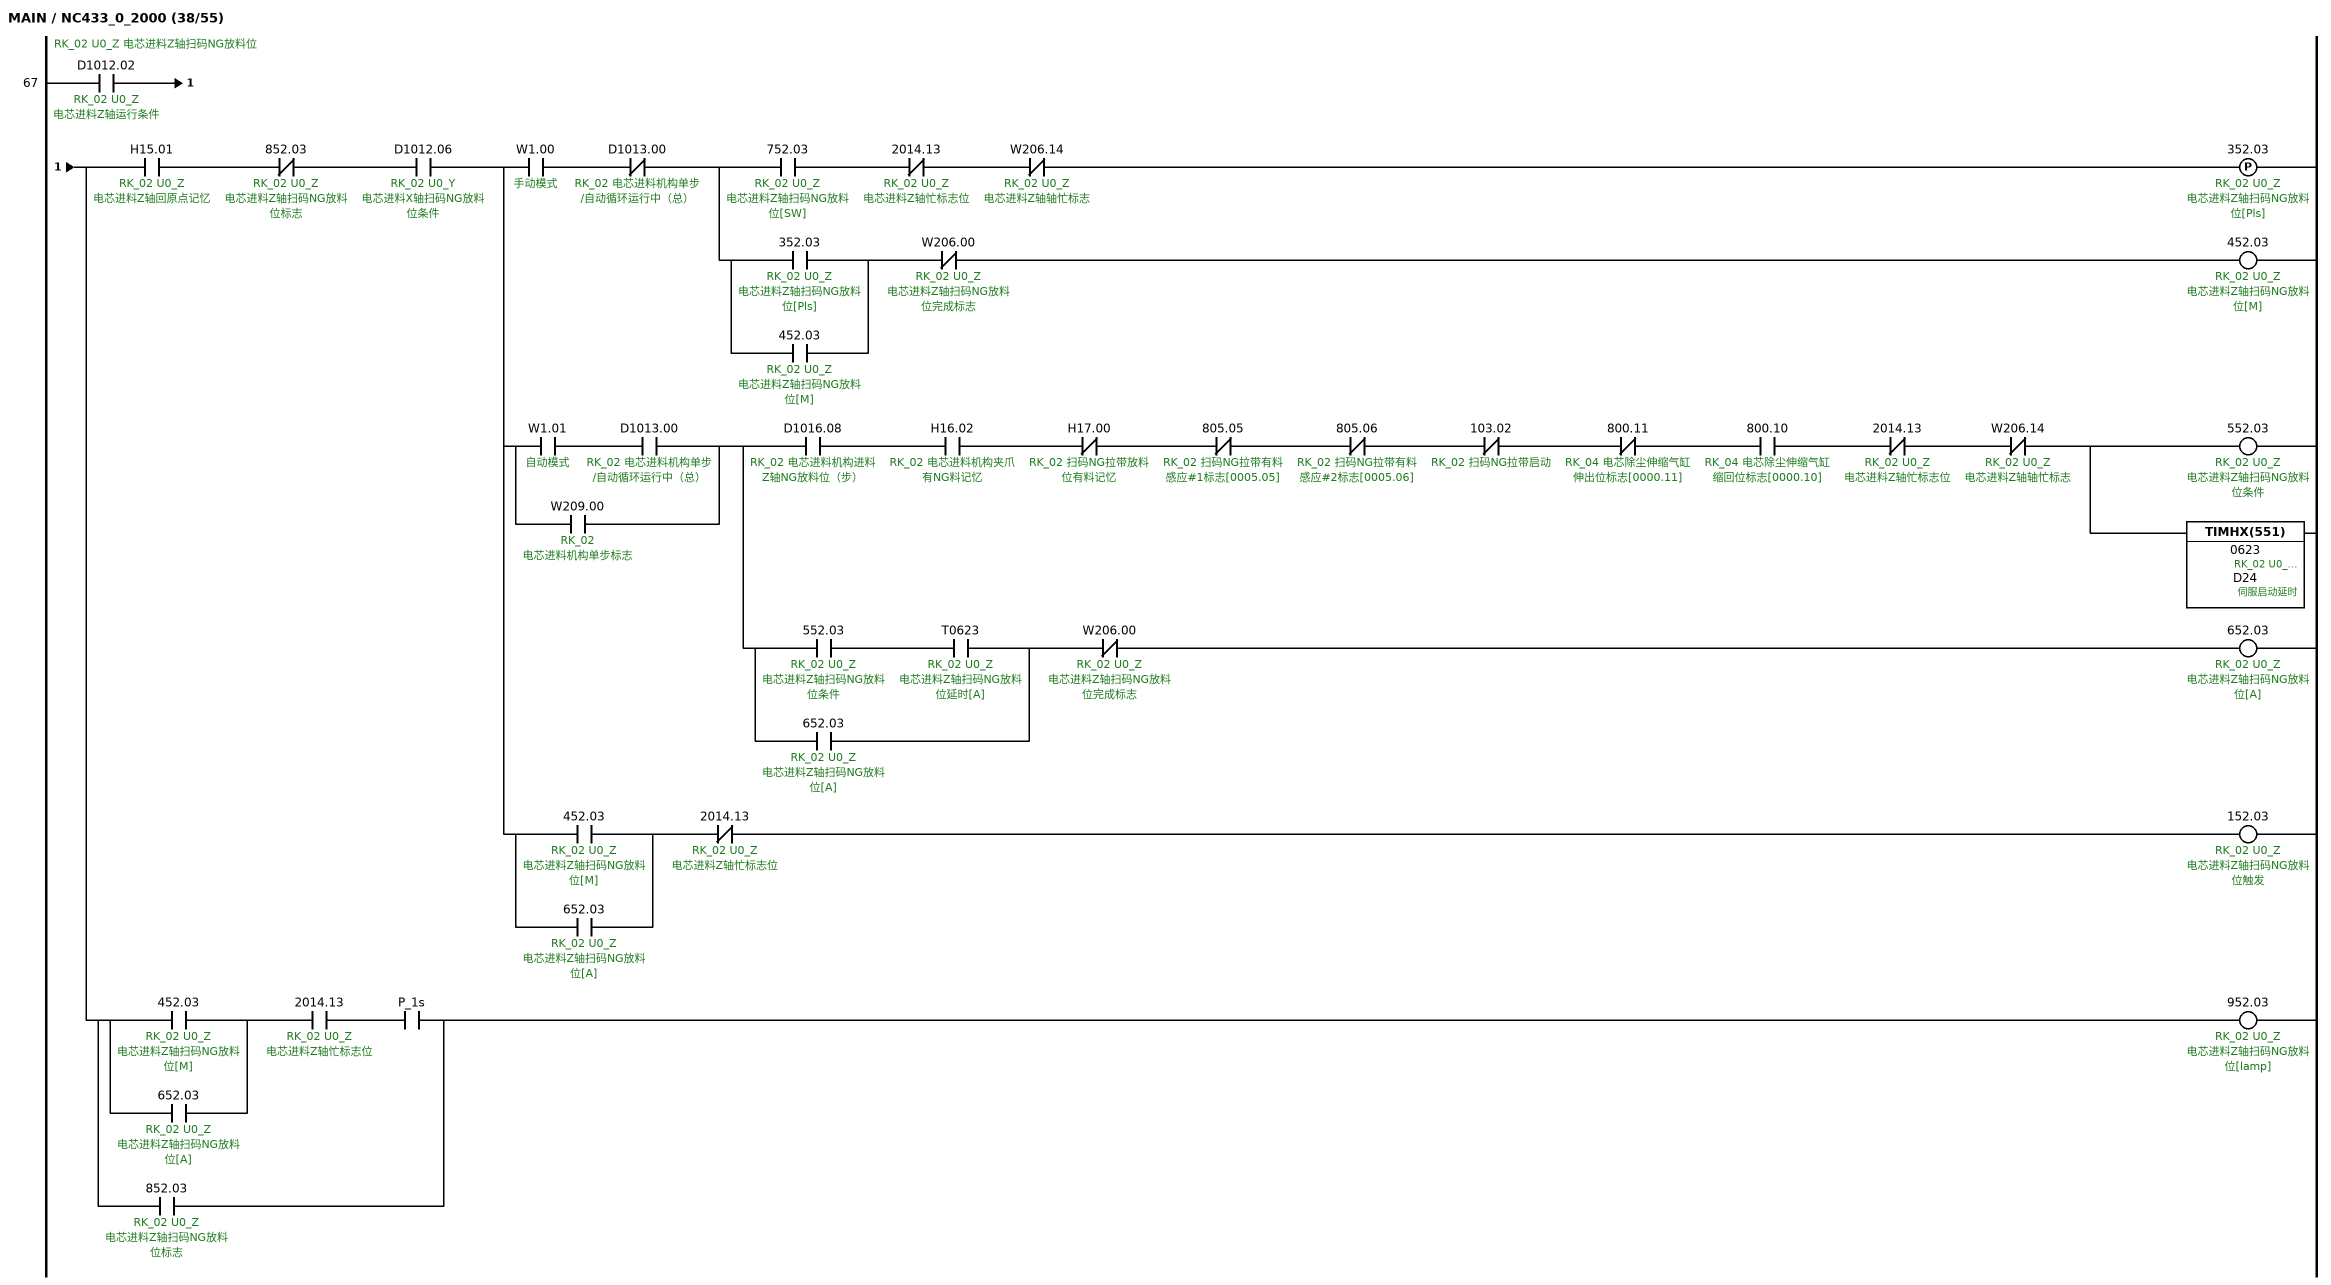
; rung 67: RK_02 U0_Z 电芯进料Z轴扫码NG放料位
LD D1012.02  ; RK_02 U0_Z 电芯进料Z轴运行条件
OUT TR0
AND H15.01  ; RK_02 U0_Z 电芯进料Z轴回原点记忆
ANDNOT 852.03  ; RK_02 U0_Z 电芯进料Z轴扫码NG放料位标志
AND D1012.06  ; RK_02 U0_Y 电芯进料X轴扫码NG放料位条件
OUT TR1
AND W1.00  ; 手动模式
ANDNOT D1013.00  ; RK_02 电芯进料机构单步/自动循环运行中（总）
OUT TR2
AND 752.03  ; RK_02 U0_Z 电芯进料Z轴扫码NG放料位[SW]
ANDNOT 2014.13  ; RK_02 U0_Z 电芯进料Z轴忙标志位
ANDNOT W206.14  ; RK_02 U0_Z 电芯进料Z轴轴忙标志
DIFU(013) 352.03  ; RK_02 U0_Z 电芯进料Z轴扫码NG放料位[Pls]
LD TR2
LD 352.03  ; RK_02 U0_Z 电芯进料Z轴扫码NG放料位[Pls]
OR 452.03  ; RK_02 U0_Z 电芯进料Z轴扫码NG放料位[M]
ANDLD
ANDNOT W206.00  ; RK_02 U0_Z 电芯进料Z轴扫码NG放料位完成标志
OUT 452.03  ; RK_02 U0_Z 电芯进料Z轴扫码NG放料位[M]
LD TR1
LD W1.01  ; 自动模式
AND D1013.00  ; RK_02 电芯进料机构单步/自动循环运行中（总）
OR W209.00  ; RK_02  电芯进料机构单步标志
ANDLD
OUT TR2
AND D1016.08  ; RK_02 电芯进料机构进料Z轴NG放料位（步）
AND H16.02  ; RK_02 电芯进料机构夹爪有NG料记忆
ANDNOT H17.00  ; RK_02 扫码NG拉带放料位有料记忆
ANDNOT 805.05  ; RK_02 扫码NG拉带有料感应#1标志[0005.05]
ANDNOT 805.06  ; RK_02 扫码NG拉带有料感应#2标志[0005.06]
ANDNOT 103.02  ; RK_02 扫码NG拉带启动
ANDNOT 800.11  ; RK_04 电芯除尘伸缩气缸伸出位标志[0000.11]
AND 800.10  ; RK_04 电芯除尘伸缩气缸缩回位标志[0000.10]
ANDNOT 2014.13  ; RK_02 U0_Z 电芯进料Z轴忙标志位
ANDNOT W206.14  ; RK_02 U0_Z 电芯进料Z轴轴忙标志
OUT 552.03  ; RK_02 U0_Z 电芯进料Z轴扫码NG放料位条件
TIMHX(551) 0623 D24  ; 伺服启动延时, RK_02 U0_Z 电芯进料Z轴扫码NG放料位延时[A]
LD TR2
LD 552.03  ; RK_02 U0_Z 电芯进料Z轴扫码NG放料位条件
AND T0623  ; RK_02 U0_Z 电芯进料Z轴扫码NG放料位延时[A]
OR 652.03  ; RK_02 U0_Z 电芯进料Z轴扫码NG放料位[A]
ANDLD
ANDNOT W206.00  ; RK_02 U0_Z 电芯进料Z轴扫码NG放料位完成标志
OUT 652.03  ; RK_02 U0_Z 电芯进料Z轴扫码NG放料位[A]
LD TR1
LD 452.03  ; RK_02 U0_Z 电芯进料Z轴扫码NG放料位[M]
OR 652.03  ; RK_02 U0_Z 电芯进料Z轴扫码NG放料位[A]
ANDLD
ANDNOT 2014.13  ; RK_02 U0_Z 电芯进料Z轴忙标志位
OUT 152.03  ; RK_02 U0_Z 电芯进料Z轴扫码NG放料位触发
LD TR0
LD 452.03  ; RK_02 U0_Z 电芯进料Z轴扫码NG放料位[M]
OR 652.03  ; RK_02 U0_Z 电芯进料Z轴扫码NG放料位[A]
AND 2014.13  ; RK_02 U0_Z 电芯进料Z轴忙标志位
AND P_1s
OR 852.03  ; RK_02 U0_Z 电芯进料Z轴扫码NG放料位标志
ANDLD
OUT 952.03  ; RK_02 U0_Z 电芯进料Z轴扫码NG放料位[lamp]

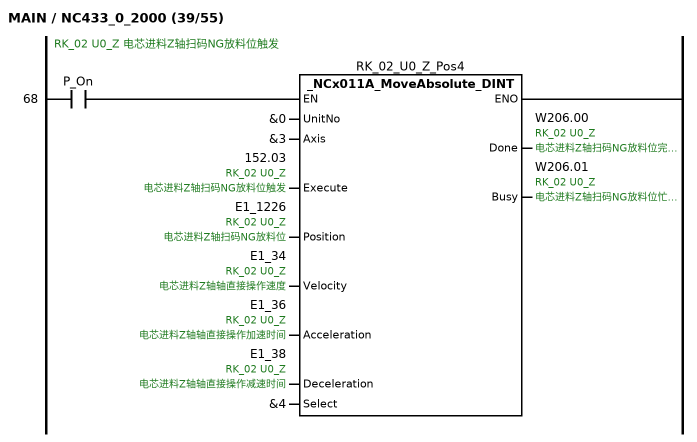
; rung 68: RK_02 U0_Z 电芯进料Z轴扫码NG放料位触发
LD P_On
CALL RK_02_U0_Z_Pos4 : _NCx011A_MoveAbsolute_DINT (UnitNo := &0, Axis := &3, Execute := 152.03, Position := E1_1226, Velocity := E1_34, Acceleration := E1_36, Deceleration := E1_38, Select := &4, Done => W206.00, Busy => W206.01)  ; RK_02 U0_Z 电芯进料Z轴扫码NG放料位触发, RK_02 U0_Z 电芯进料Z轴扫码NG放料位, RK_02 U0_Z 电芯进料Z轴轴直接操作速度, RK_02 U0_Z 电芯进料Z轴轴直接操作加速时间, RK_02 U0_Z 电芯进料Z轴轴直接操作减速时间, RK_02 U0_Z 电芯进料Z轴扫码NG放料位完成标志, RK_02 U0_Z 电芯进料Z轴扫码NG放料位忙标志

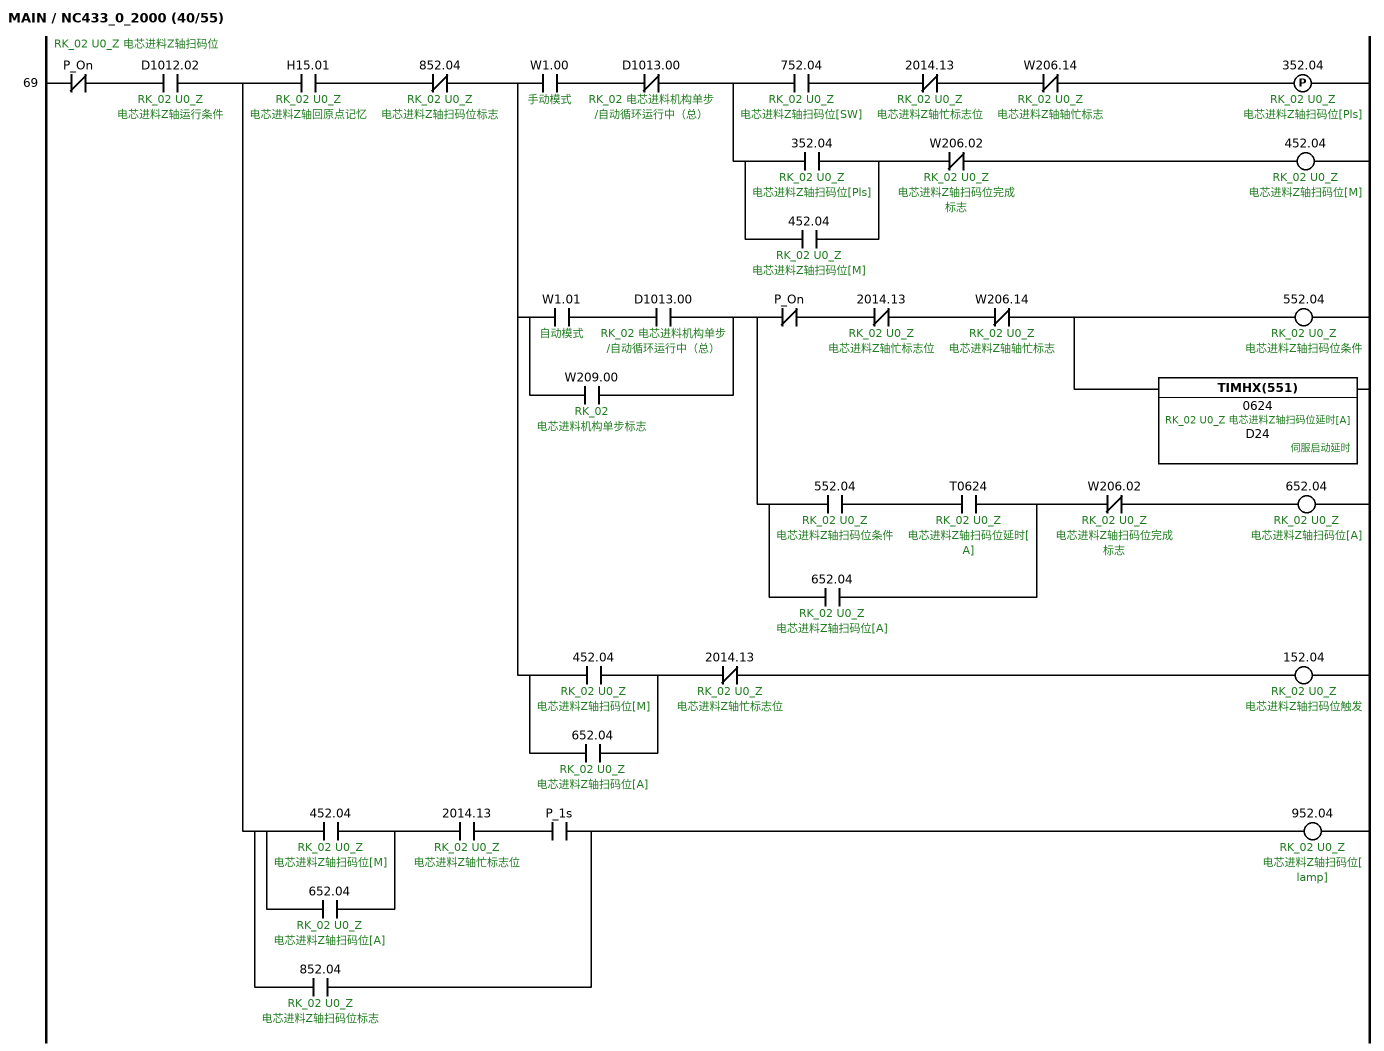
; rung 69: RK_02 U0_Z 电芯进料Z轴扫码位
LDNOT P_On
AND D1012.02  ; RK_02 U0_Z 电芯进料Z轴运行条件
OUT TR0
AND H15.01  ; RK_02 U0_Z 电芯进料Z轴回原点记忆
ANDNOT 852.04  ; RK_02 U0_Z 电芯进料Z轴扫码位标志
OUT TR1
AND W1.00  ; 手动模式
ANDNOT D1013.00  ; RK_02 电芯进料机构单步/自动循环运行中（总）
OUT TR2
AND 752.04  ; RK_02 U0_Z 电芯进料Z轴扫码位[SW]
ANDNOT 2014.13  ; RK_02 U0_Z 电芯进料Z轴忙标志位
ANDNOT W206.14  ; RK_02 U0_Z 电芯进料Z轴轴忙标志
DIFU(013) 352.04  ; RK_02 U0_Z 电芯进料Z轴扫码位[Pls]
LD TR2
LD 352.04  ; RK_02 U0_Z 电芯进料Z轴扫码位[Pls]
OR 452.04  ; RK_02 U0_Z 电芯进料Z轴扫码位[M]
ANDLD
ANDNOT W206.02  ; RK_02 U0_Z 电芯进料Z轴扫码位完成标志
OUT 452.04  ; RK_02 U0_Z 电芯进料Z轴扫码位[M]
LD TR1
LD W1.01  ; 自动模式
AND D1013.00  ; RK_02 电芯进料机构单步/自动循环运行中（总）
OR W209.00  ; RK_02  电芯进料机构单步标志
ANDLD
OUT TR2
ANDNOT P_On  // RK_02 U0_Z 电芯进料Z轴扫码位（步）
ANDNOT 2014.13  ; RK_02 U0_Z 电芯进料Z轴忙标志位
ANDNOT W206.14  ; RK_02 U0_Z 电芯进料Z轴轴忙标志
OUT 552.04  ; RK_02 U0_Z 电芯进料Z轴扫码位条件
TIMHX(551) 0624 D24  ; 伺服启动延时, RK_02 U0_Z 电芯进料Z轴扫码位延时[A]
LD TR2
LD 552.04  ; RK_02 U0_Z 电芯进料Z轴扫码位条件
AND T0624  ; RK_02 U0_Z 电芯进料Z轴扫码位延时[A]
OR 652.04  ; RK_02 U0_Z 电芯进料Z轴扫码位[A]
ANDLD
ANDNOT W206.02  ; RK_02 U0_Z 电芯进料Z轴扫码位完成标志
OUT 652.04  ; RK_02 U0_Z 电芯进料Z轴扫码位[A]
LD TR1
LD 452.04  ; RK_02 U0_Z 电芯进料Z轴扫码位[M]
OR 652.04  ; RK_02 U0_Z 电芯进料Z轴扫码位[A]
ANDLD
ANDNOT 2014.13  ; RK_02 U0_Z 电芯进料Z轴忙标志位
OUT 152.04  ; RK_02 U0_Z 电芯进料Z轴扫码位触发
LD TR0
LD 452.04  ; RK_02 U0_Z 电芯进料Z轴扫码位[M]
OR 652.04  ; RK_02 U0_Z 电芯进料Z轴扫码位[A]
AND 2014.13  ; RK_02 U0_Z 电芯进料Z轴忙标志位
AND P_1s
OR 852.04  ; RK_02 U0_Z 电芯进料Z轴扫码位标志
ANDLD
OUT 952.04  ; RK_02 U0_Z 电芯进料Z轴扫码位[lamp]

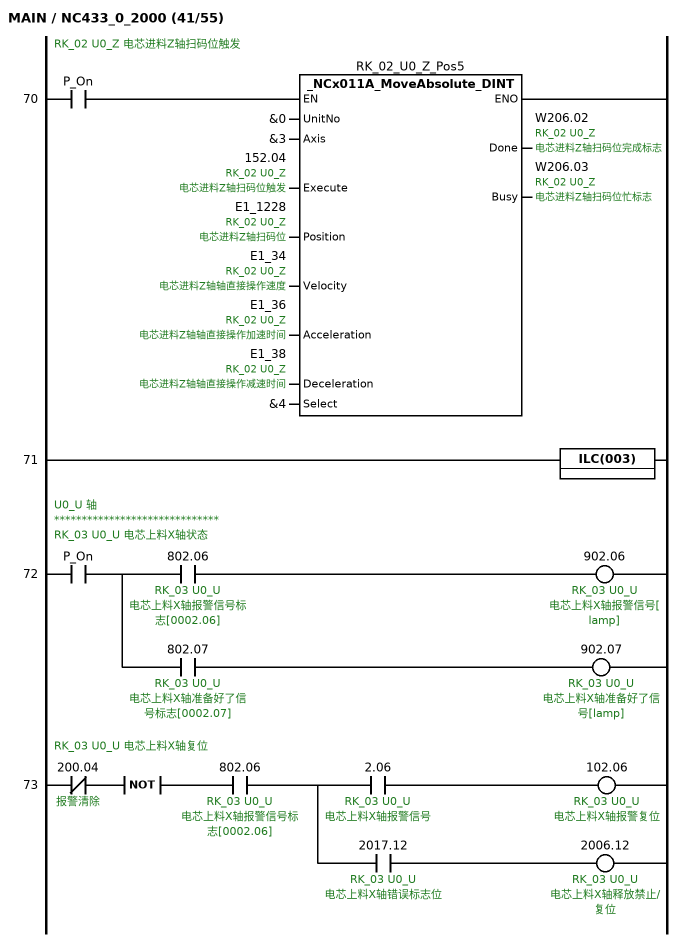
; rung 70: RK_02 U0_Z 电芯进料Z轴扫码位触发
LD P_On
CALL RK_02_U0_Z_Pos5 : _NCx011A_MoveAbsolute_DINT (UnitNo := &0, Axis := &3, Execute := 152.04, Position := E1_1228, Velocity := E1_34, Acceleration := E1_36, Deceleration := E1_38, Select := &4, Done => W206.02, Busy => W206.03)  ; RK_02 U0_Z 电芯进料Z轴扫码位触发, RK_02 U0_Z 电芯进料Z轴扫码位, RK_02 U0_Z 电芯进料Z轴轴直接操作速度, RK_02 U0_Z 电芯进料Z轴轴直接操作加速时间, RK_02 U0_Z 电芯进料Z轴轴直接操作减速时间, RK_02 U0_Z 电芯进料Z轴扫码位完成标志, RK_02 U0_Z 电芯进料Z轴扫码位忙标志
; rung 71
ILC(003)
; rung 72: U0_U 轴 / ****************************** / RK_03 U0_U 电芯上料X轴状态
LD P_On
OUT TR0
AND 802.06  ; RK_03 U0_U 电芯上料X轴报警信号标志[0002.06]
OUT 902.06  ; RK_03 U0_U 电芯上料X轴报警信号[lamp]
LD TR0
AND 802.07  ; RK_03 U0_U 电芯上料X轴准备好了信号标志[0002.07]
OUT 902.07  ; RK_03 U0_U 电芯上料X轴准备好了信号[lamp]
; rung 73: RK_03 U0_U 电芯上料X轴复位
LDNOT 200.04  ; 报警清除
NOT(520)
AND 802.06  ; RK_03 U0_U 电芯上料X轴报警信号标志[0002.06]
OUT TR0
AND 2.06  ; RK_03 U0_U 电芯上料X轴报警信号
OUT 102.06  ; RK_03 U0_U 电芯上料X轴报警复位
LD TR0
AND 2017.12  ; RK_03 U0_U 电芯上料X轴错误标志位
OUT 2006.12  ; RK_03 U0_U 电芯上料X轴释放禁止/复位

